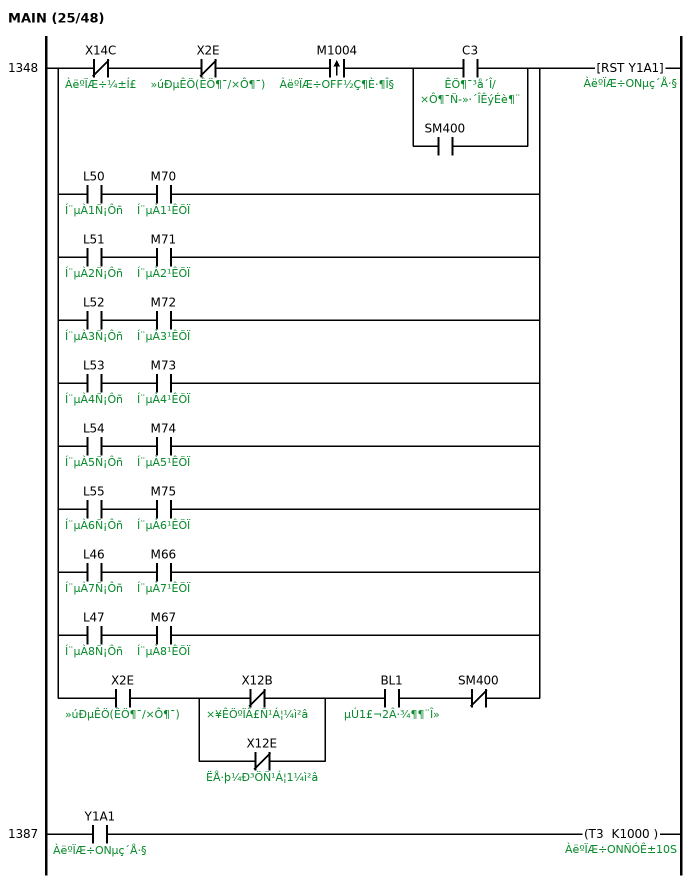
[picture p24: ladder of MAIN, rungs at steps 1348 to 1387]
1348  LDI     X14C  ; ÀëºÏÆ÷¼±Í£
      ANI     X2E  ; »úÐµÊÖ(ÊÖ¶¯/×Ô¶¯)
      ANDP    M1004  ; ÀëºÏÆ÷OFF½Ç¶È·¶Î§
      LD      C3  ; ÊÖ¶¯³å´Î/×Ô¶¯Ñ­»·´ÎÊýÉè¶¨
      OR      SM400
      ANB
      LD      L50  ; Í¨µÀ1Ñ¡Ôñ
      AND     M70  ; Í¨µÀ1¹ÊÕÏ
      ORB
      LD      L51  ; Í¨µÀ2Ñ¡Ôñ
      AND     M71  ; Í¨µÀ2¹ÊÕÏ
      ORB
      LD      L52  ; Í¨µÀ3Ñ¡Ôñ
      AND     M72  ; Í¨µÀ3¹ÊÕÏ
      ORB
      LD      L53  ; Í¨µÀ4Ñ¡Ôñ
      AND     M73  ; Í¨µÀ4¹ÊÕÏ
      ORB
      LD      L54  ; Í¨µÀ5Ñ¡Ôñ
      AND     M74  ; Í¨µÀ5¹ÊÕÏ
      ORB
      LD      L55  ; Í¨µÀ6Ñ¡Ôñ
      AND     M75  ; Í¨µÀ6¹ÊÕÏ
      ORB
      LD      L46  ; Í¨µÀ7Ñ¡Ôñ
      AND     M66  ; Í¨µÀ7¹ÊÕÏ
      ORB
      LD      L47  ; Í¨µÀ8Ñ¡Ôñ
      AND     M67  ; Í¨µÀ8¹ÊÕÏ
      ORB
      LD      X2E  ; »úÐµÊÖ(ÊÖ¶¯/×Ô¶¯)
      LDI     X12B  ; ×¥ÊÖºÏÂ£Ñ¹Á¦¼ì²â
      ORI     X12E  ; ËÅ·þ¼Ð³ÖÑ¹Á¦1¼ì²â
      ANB
      AND     BL1  ; µÚ1£¬2Â·¾¶¶¨Î»
      ANI     SM400
      ORB
      RST     Y1A1  ; ÀëºÏÆ÷ONµç´Å·§
1387  LD      Y1A1  ; ÀëºÏÆ÷ONµç´Å·§
      OUT     T3 K1000  ; ÀëºÏÆ÷ONÑÓÊ±10S
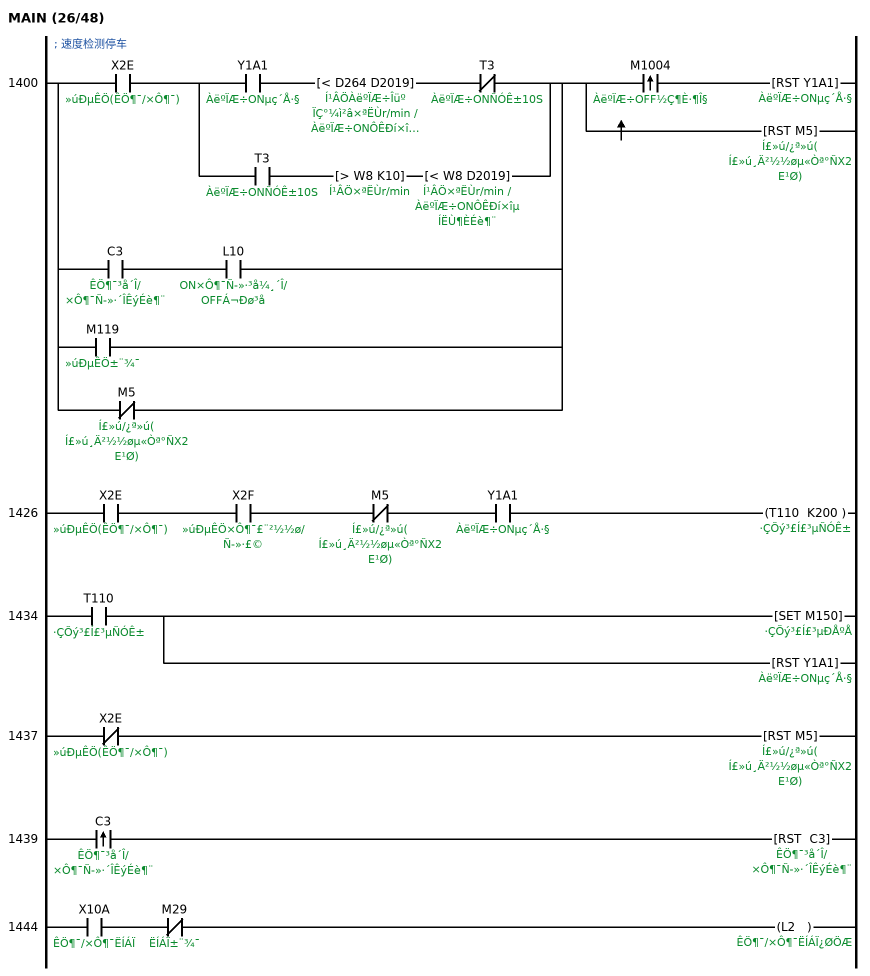
; 速度检测停车
1400  LD      X2E  ; »úÐµÊÖ(ÊÖ¶¯/×Ô¶¯)
      LD      Y1A1  ; ÀëºÏÆ÷ONµç´Å·§
      AND<    D264 D2019  ; Í¹ÂÖÀëºÏÆ÷ÎüºÏÇ°¼ì²â×ªËÙr/min / ÀëºÏÆ÷ONÔÊÐí×îµÍËÙ¶ÈÉè¶¨
      ANI     T3  ; ÀëºÏÆ÷ONÑÓÊ±10S
      LD      T3  ; ÀëºÏÆ÷ONÑÓÊ±10S
      AND>    W8 K10  ; Í¹ÂÖ×ªËÙr/min
      AND<    W8 D2019  ; Í¹ÂÖ×ªËÙr/min / ÀëºÏÆ÷ONÔÊÐí×îµÍËÙ¶ÈÉè¶¨
      ORB
      ANB
      LD      C3  ; ÊÖ¶¯³å´Î/×Ô¶¯Ñ­»·´ÎÊýÉè¶¨
      AND     L10  ; ON×Ô¶¯Ñ­»·³å¼¸´Î/OFFÁ¬Ðø³å
      ORB
      OR      M119  ; »úÐµÊÖ±¨¾¯
      ORI     M5  ; Í£»ú/¿ª»ú(Í£»ú¸Ä²½½øµ«Òª°ÑX2E¹Ø)
      MPS
      ANDP    M1004  ; ÀëºÏÆ÷OFF½Ç¶È·¶Î§
      RST     Y1A1  ; ÀëºÏÆ÷ONµç´Å·§
      MPP
      MEP
      RST     M5  ; Í£»ú/¿ª»ú(Í£»ú¸Ä²½½øµ«Òª°ÑX2E¹Ø)
1426  LD      X2E  ; »úÐµÊÖ(ÊÖ¶¯/×Ô¶¯)
      AND     X2F  ; »úÐµÊÖ×Ô¶¯£¨²½½ø/Ñ­»·£©
      ANI     M5  ; Í£»ú/¿ª»ú(Í£»ú¸Ä²½½øµ«Òª°ÑX2E¹Ø)
      AND     Y1A1  ; ÀëºÏÆ÷ONµç´Å·§
      OUT     T110 K200  ; ·ÇÕý³£Í£³µÑÓÊ±
1434  LD      T110  ; ·ÇÕý³£Í£³µÑÓÊ±
      SET     M150  ; ·ÇÕý³£Í£³µÐÅºÅ
      RST     Y1A1  ; ÀëºÏÆ÷ONµç´Å·§
1437  LDI     X2E  ; »úÐµÊÖ(ÊÖ¶¯/×Ô¶¯)
      RST     M5  ; Í£»ú/¿ª»ú(Í£»ú¸Ä²½½øµ«Òª°ÑX2E¹Ø)
1439  LDP     C3  ; ÊÖ¶¯³å´Î/×Ô¶¯Ñ­»·´ÎÊýÉè¶¨
      RST     C3  ; ÊÖ¶¯³å´Î/×Ô¶¯Ñ­»·´ÎÊýÉè¶¨
1444  LD      X10A  ; ÊÖ¶¯/×Ô¶¯ËÍÁÏ
      ANI     M29  ; ËÍÁÏ±¨¾¯
      OUT     L2  ; ÊÖ¶¯/×Ô¶¯ËÍÁÏ¿ØÖÆ
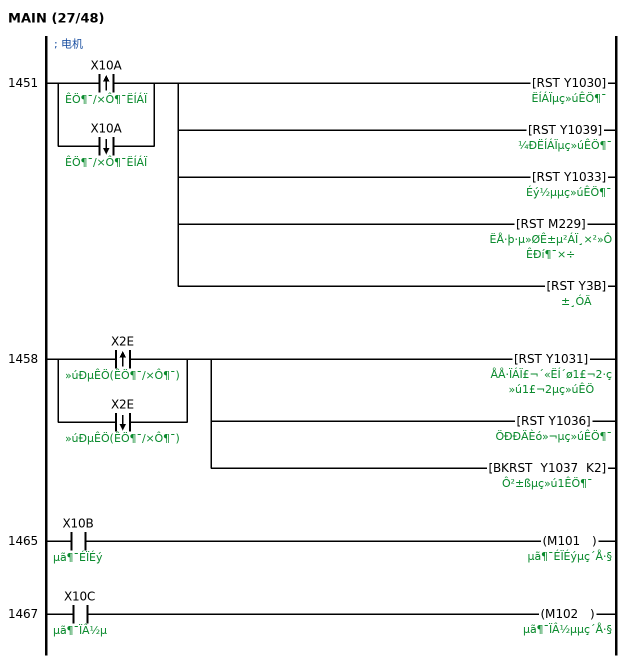
; 电机
1451  LDP     X10A  ; ÊÖ¶¯/×Ô¶¯ËÍÁÏ
      ORF     X10A  ; ÊÖ¶¯/×Ô¶¯ËÍÁÏ
      RST     Y1030  ; ËÍÁÏµç»úÊÖ¶¯
      RST     Y1039  ; ¼ÐËÍÁÏµç»úÊÖ¶¯
      RST     Y1033  ; Éý½µµç»úÊÖ¶¯
      RST     M229  ; ËÅ·þ·µ»ØÊ±µ²ÁÏ¸×²»ÔÊÐí¶¯×÷
      RST     Y3B  ; ±¸ÓÃ
1458  LDP     X2E  ; »úÐµÊÖ(ÊÖ¶¯/×Ô¶¯)
      ORF     X2E  ; »úÐµÊÖ(ÊÖ¶¯/×Ô¶¯)
      RST     Y1031  ; ÅÅ·ÏÁÏ£¬´«ËÍ´ø1£¬2·ç»ú1£¬2µç»úÊÖ
      RST     Y1036  ; ÖÐÐÄÈó»¬µç»úÊÖ¶¯
      BKRST   Y1037 K2  ; Ô²±ßµç»ú1ÊÖ¶¯
1465  LD      X10B  ; µã¶¯ÉÏÉý
      OUT     M101  ; µã¶¯ÉÏÉýµç´Å·§
1467  LD      X10C  ; µã¶¯ÏÂ½µ
      OUT     M102  ; µã¶¯ÏÂ½µµç´Å·§
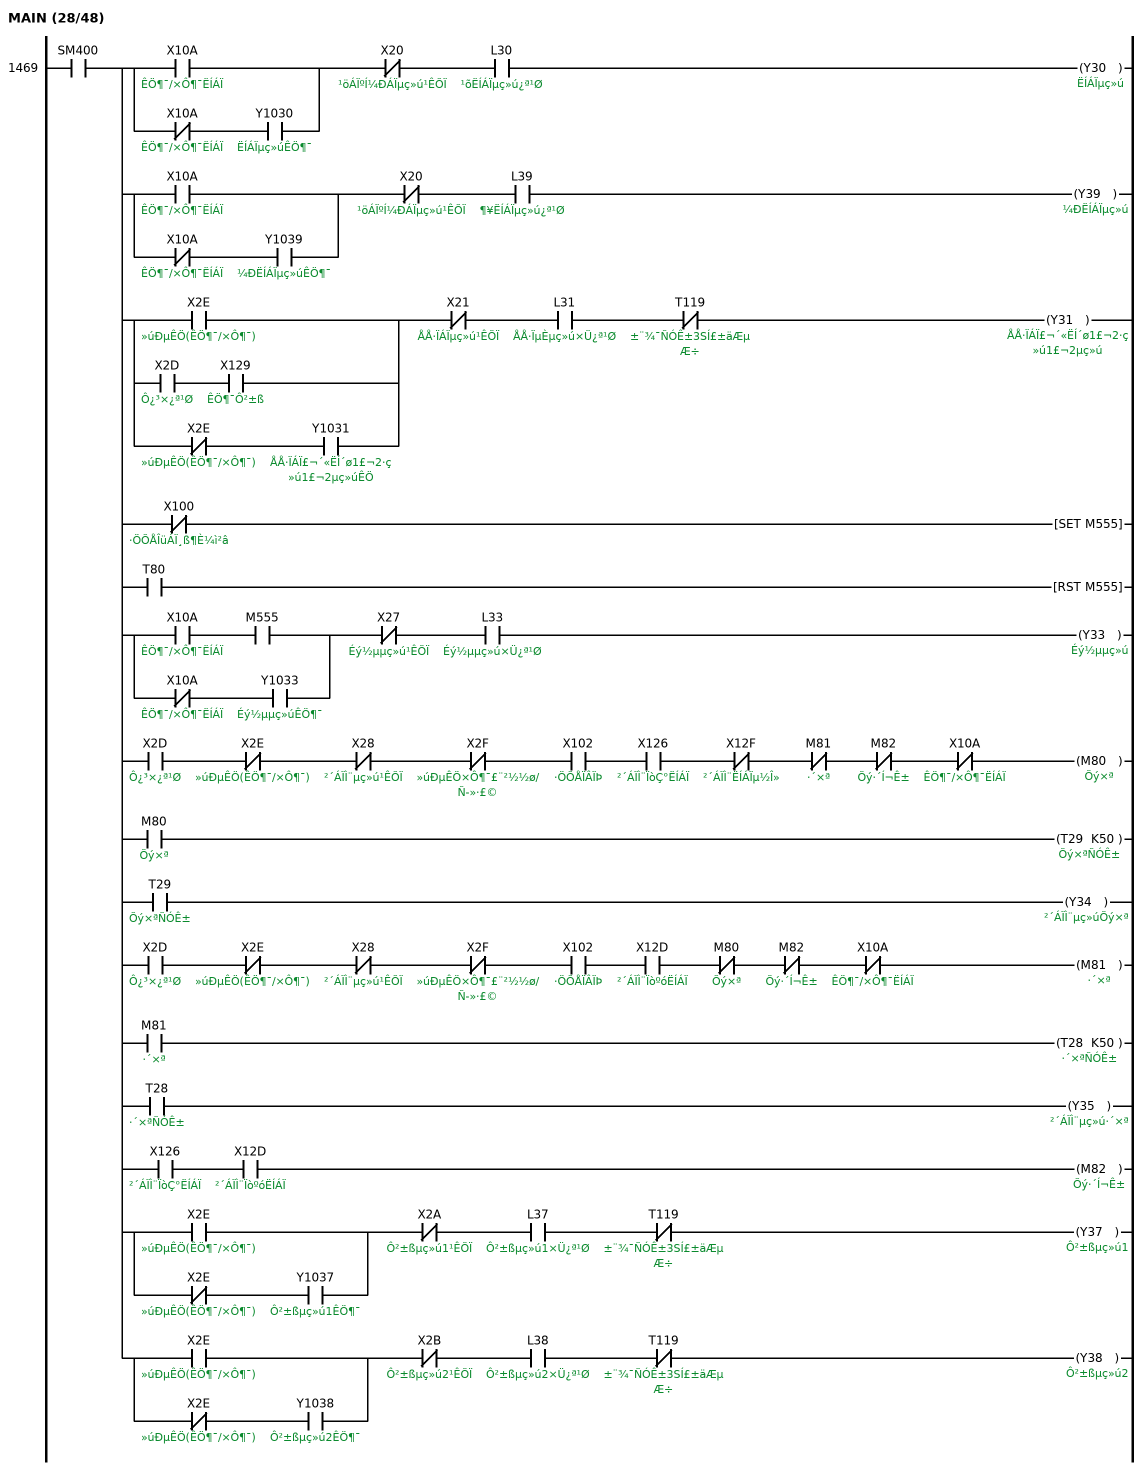
1469  LD      SM400
      MPS
      LD      X10A  ; ÊÖ¶¯/×Ô¶¯ËÍÁÏ
      LDI     X10A  ; ÊÖ¶¯/×Ô¶¯ËÍÁÏ
      AND     Y1030  ; ËÍÁÏµç»úÊÖ¶¯
      ORB
      ANB
      ANI     X20  ; ¹öÁÏºÍ¼ÐÁÏµç»ú¹ÊÕÏ
      AND     L30  ; ¹õËÍÁÏµç»ú¿ª¹Ø
      OUT     Y30  ; ËÍÁÏµç»ú
      MRD
      LD      X10A  ; ÊÖ¶¯/×Ô¶¯ËÍÁÏ
      LDI     X10A  ; ÊÖ¶¯/×Ô¶¯ËÍÁÏ
      AND     Y1039  ; ¼ÐËÍÁÏµç»úÊÖ¶¯
      ORB
      ANB
      ANI     X20  ; ¹öÁÏºÍ¼ÐÁÏµç»ú¹ÊÕÏ
      AND     L39  ; ¶¥ËÍÁÏµç»ú¿ª¹Ø
      OUT     Y39  ; ¼ÐËÍÁÏµç»ú
      MRD
      LD      X2E  ; »úÐµÊÖ(ÊÖ¶¯/×Ô¶¯)
      LD      X2D  ; Ô¿³×¿ª¹Ø
      AND     X129  ; ÊÖ¶¯Ô²±ß
      ORB
      LDI     X2E  ; »úÐµÊÖ(ÊÖ¶¯/×Ô¶¯)
      AND     Y1031  ; ÅÅ·ÏÁÏ£¬´«ËÍ´ø1£¬2·ç»ú1£¬2µç»úÊÖ
      ORB
      ANB
      ANI     X21  ; ÅÅ·ÏÁÏµç»ú¹ÊÕÏ
      AND     L31  ; ÅÅ·ÏµÈµç»ú×Ü¿ª¹Ø
      ANI     T119  ; ±¨¾¯ÑÓÊ±3SÍ£±äÆµÆ÷
      OUT     Y31  ; ÅÅ·ÏÁÏ£¬´«ËÍ´ø1£¬2·ç»ú1£¬2µç»ú
      MRD
      ANI     X100  ; ·ÖÕÅÎüÁÏ¸ß¶È¼ì²â
      SET     M555
      MRD
      AND     T80
      RST     M555
      MRD
      LD      X10A  ; ÊÖ¶¯/×Ô¶¯ËÍÁÏ
      AND     M555
      LDI     X10A  ; ÊÖ¶¯/×Ô¶¯ËÍÁÏ
      AND     Y1033  ; Éý½µµç»úÊÖ¶¯
      ORB
      ANB
      ANI     X27  ; Éý½µµç»ú¹ÊÕÏ
      AND     L33  ; Éý½µµç»ú×Ü¿ª¹Ø
      OUT     Y33  ; Éý½µµç»ú
      MRD
      AND     X2D  ; Ô¿³×¿ª¹Ø
      ANI     X2E  ; »úÐµÊÖ(ÊÖ¶¯/×Ô¶¯)
      ANI     X28  ; ²´ÁÏÌ¨µç»ú¹ÊÕÏ
      ANI     X2F  ; »úÐµÊÖ×Ô¶¯£¨²½½ø/Ñ­»·£©
      AND     X102  ; ·ÖÕÅÏÂÏÞ
      AND     X126  ; ²´ÁÏÌ¨ÏòÇ°ËÍÁÏ
      ANI     X12F  ; ²´ÁÏÌ¨ËÍÁÏµ½Î»
      ANI     M81  ; ·´×ª
      ANI     M82  ; Õý·´Í¬Ê±
      ANI     X10A  ; ÊÖ¶¯/×Ô¶¯ËÍÁÏ
      OUT     M80  ; Õý×ª
      MRD
      AND     M80  ; Õý×ª
      OUT     T29 K50  ; Õý×ªÑÓÊ±
      MRD
      AND     T29  ; Õý×ªÑÓÊ±
      OUT     Y34  ; ²´ÁÏÌ¨µç»úÕý×ª
      MRD
      AND     X2D  ; Ô¿³×¿ª¹Ø
      ANI     X2E  ; »úÐµÊÖ(ÊÖ¶¯/×Ô¶¯)
      ANI     X28  ; ²´ÁÏÌ¨µç»ú¹ÊÕÏ
      ANI     X2F  ; »úÐµÊÖ×Ô¶¯£¨²½½ø/Ñ­»·£©
      AND     X102  ; ·ÖÕÅÏÂÏÞ
      AND     X12D  ; ²´ÁÏÌ¨ÏòºóËÍÁÏ
      ANI     M80  ; Õý×ª
      ANI     M82  ; Õý·´Í¬Ê±
      ANI     X10A  ; ÊÖ¶¯/×Ô¶¯ËÍÁÏ
      OUT     M81  ; ·´×ª
      MRD
      AND     M81  ; ·´×ª
      OUT     T28 K50  ; ·´×ªÑÓÊ±
      MRD
      AND     T28  ; ·´×ªÑÓÊ±
      OUT     Y35  ; ²´ÁÏÌ¨µç»ú·´×ª
      MRD
      AND     X126  ; ²´ÁÏÌ¨ÏòÇ°ËÍÁÏ
      AND     X12D  ; ²´ÁÏÌ¨ÏòºóËÍÁÏ
      OUT     M82  ; Õý·´Í¬Ê±
      MRD
      LD      X2E  ; »úÐµÊÖ(ÊÖ¶¯/×Ô¶¯)
      LDI     X2E  ; »úÐµÊÖ(ÊÖ¶¯/×Ô¶¯)
      AND     Y1037  ; Ô²±ßµç»ú1ÊÖ¶¯
      ORB
      ANB
      ANI     X2A  ; Ô²±ßµç»ú1¹ÊÕÏ
      AND     L37  ; Ô²±ßµç»ú1×Ü¿ª¹Ø
      ANI     T119  ; ±¨¾¯ÑÓÊ±3SÍ£±äÆµÆ÷
      OUT     Y37  ; Ô²±ßµç»ú1
      MPP
      LD      X2E  ; »úÐµÊÖ(ÊÖ¶¯/×Ô¶¯)
      LDI     X2E  ; »úÐµÊÖ(ÊÖ¶¯/×Ô¶¯)
      AND     Y1038  ; Ô²±ßµç»ú2ÊÖ¶¯
      ORB
      ANB
      ANI     X2B  ; Ô²±ßµç»ú2¹ÊÕÏ
      AND     L38  ; Ô²±ßµç»ú2×Ü¿ª¹Ø
      ANI     T119  ; ±¨¾¯ÑÓÊ±3SÍ£±äÆµÆ÷
      OUT     Y38  ; Ô²±ßµç»ú2
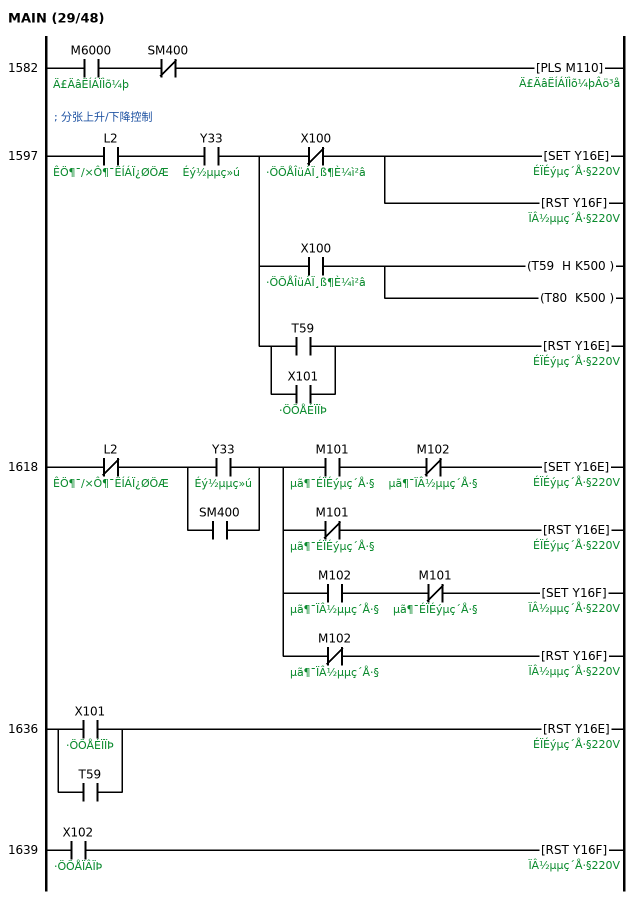
1582  LD      M6000  ; Ä£ÄâËÍÁÏÌõ¼þ
      ANI     SM400
      PLS     M110  ; Ä£ÄâËÍÁÏÌõ¼þÂö³å
; 分张上升/下降控制
1597  LD      L2  ; ÊÖ¶¯/×Ô¶¯ËÍÁÏ¿ØÖÆ
      AND     Y33  ; Éý½µµç»ú
      MPS
      ANI     X100  ; ·ÖÕÅÎüÁÏ¸ß¶È¼ì²â
      SET     Y16E  ; ÉÏÉýµç´Å·§220V
      RST     Y16F  ; ÏÂ½µµç´Å·§220V
      MRD
      AND     X100  ; ·ÖÕÅÎüÁÏ¸ß¶È¼ì²â
      OUTH    T59 K500
      OUT     T80 K500
      MPP
      LD      T59
      OR      X101  ; ·ÖÕÅÉÏÏÞ
      ANB
      RST     Y16E  ; ÉÏÉýµç´Å·§220V
1618  LDI     L2  ; ÊÖ¶¯/×Ô¶¯ËÍÁÏ¿ØÖÆ
      LD      Y33  ; Éý½µµç»ú
      OR      SM400
      ANB
      MPS
      AND     M101  ; µã¶¯ÉÏÉýµç´Å·§
      ANI     M102  ; µã¶¯ÏÂ½µµç´Å·§
      SET     Y16E  ; ÉÏÉýµç´Å·§220V
      MRD
      ANI     M101  ; µã¶¯ÉÏÉýµç´Å·§
      RST     Y16E  ; ÉÏÉýµç´Å·§220V
      MRD
      AND     M102  ; µã¶¯ÏÂ½µµç´Å·§
      ANI     M101  ; µã¶¯ÉÏÉýµç´Å·§
      SET     Y16F  ; ÏÂ½µµç´Å·§220V
      MPP
      ANI     M102  ; µã¶¯ÏÂ½µµç´Å·§
      RST     Y16F  ; ÏÂ½µµç´Å·§220V
1636  LD      X101  ; ·ÖÕÅÉÏÏÞ
      OR      T59
      RST     Y16E  ; ÉÏÉýµç´Å·§220V
1639  LD      X102  ; ·ÖÕÅÏÂÏÞ
      RST     Y16F  ; ÏÂ½µµç´Å·§220V
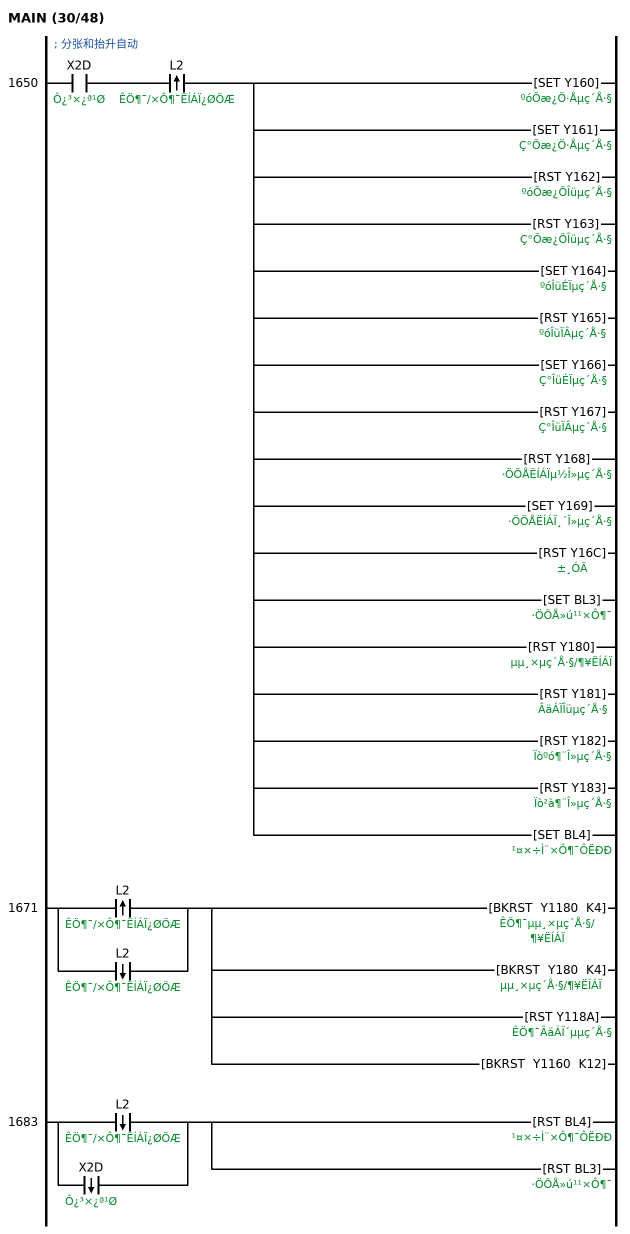
; 分张和抬升自动
1650  LD      X2D  ; Ô¿³×¿ª¹Ø
      ANDP    L2  ; ÊÖ¶¯/×Ô¶¯ËÍÁÏ¿ØÖÆ
      SET     Y160  ; ºóÕæ¿Õ·Åµç´Å·§
      SET     Y161  ; Ç°Õæ¿Õ·Åµç´Å·§
      RST     Y162  ; ºóÕæ¿ÕÎüµç´Å·§
      RST     Y163  ; Ç°Õæ¿ÕÎüµç´Å·§
      SET     Y164  ; ºóÎüÉÏµç´Å·§
      RST     Y165  ; ºóÎüÏÂµç´Å·§
      SET     Y166  ; Ç°ÎüÉÏµç´Å·§
      RST     Y167  ; Ç°ÎüÏÂµç´Å·§
      RST     Y168  ; ·ÖÕÅËÍÁÏµ½Î»µç´Å·§
      SET     Y169  ; ·ÖÕÅËÍÁÏ¸´Î»µç´Å·§
      RST     Y16C  ; ±¸ÓÃ
      SET     BL3  ; ·ÖÕÅ»ú¹¹×Ô¶¯
      RST     Y180  ; µµ¸×µç´Å·§/¶¥ËÍÁÏ
      RST     Y181  ; ÂäÁÏÎüµç´Å·§
      RST     Y182  ; Ïòºó¶¨Î»µç´Å·§
      RST     Y183  ; Ïò²à¶¨Î»µç´Å·§
      SET     BL4  ; ¹¤×÷Ì¨×Ô¶¯ÔËÐÐ
1671  LDP     L2  ; ÊÖ¶¯/×Ô¶¯ËÍÁÏ¿ØÖÆ
      ORF     L2  ; ÊÖ¶¯/×Ô¶¯ËÍÁÏ¿ØÖÆ
      BKRST   Y1180 K4  ; ÊÖ¶¯µµ¸×µç´Å·§/¶¥ËÍÁÏ
      BKRST   Y180 K4
      RST     Y118A  ; ÊÖ¶¯ÂäÁÏ´µµç´Å·§
      BKRST   Y1160 K12
1683  LDF     L2  ; ÊÖ¶¯/×Ô¶¯ËÍÁÏ¿ØÖÆ
      ORF     X2D  ; Ô¿³×¿ª¹Ø
      RST     BL4  ; ¹¤×÷Ì¨×Ô¶¯ÔËÐÐ
      RST     BL3  ; ·ÖÕÅ»ú¹¹×Ô¶¯
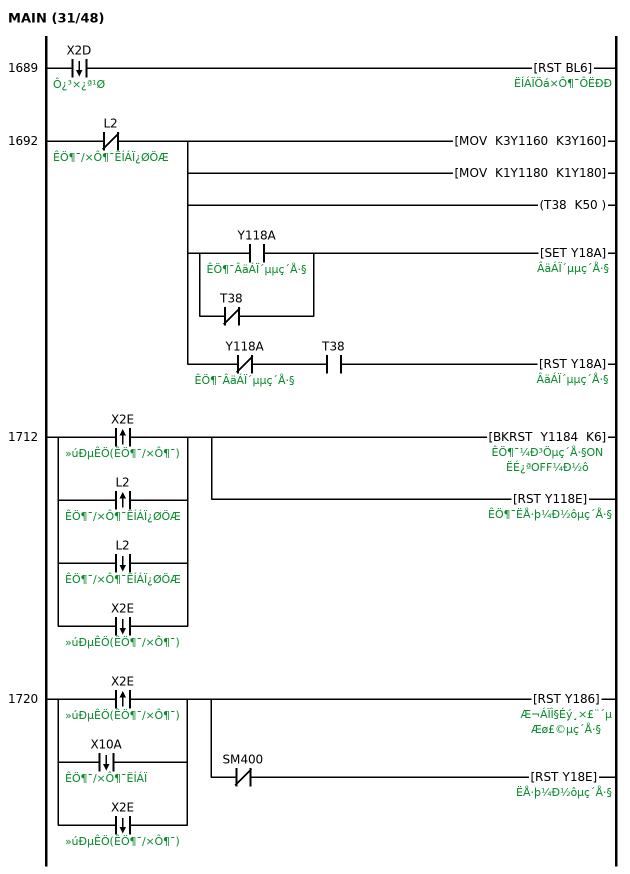
1689  LDF     X2D  ; Ô¿³×¿ª¹Ø
      RST     BL6  ; ËÍÁÏÖá×Ô¶¯ÔËÐÐ
1692  LDI     L2  ; ÊÖ¶¯/×Ô¶¯ËÍÁÏ¿ØÖÆ
      MOV     K3Y1160 K3Y160
      MOV     K1Y1180 K1Y180
      OUT     T38 K50
      MPS
      LD      Y118A  ; ÊÖ¶¯ÂäÁÏ´µµç´Å·§
      ORI     T38
      ANB
      SET     Y18A  ; ÂäÁÏ´µµç´Å·§
      MPP
      ANI     Y118A  ; ÊÖ¶¯ÂäÁÏ´µµç´Å·§
      AND     T38
      RST     Y18A  ; ÂäÁÏ´µµç´Å·§
1712  LDP     X2E  ; »úÐµÊÖ(ÊÖ¶¯/×Ô¶¯)
      ORP     L2  ; ÊÖ¶¯/×Ô¶¯ËÍÁÏ¿ØÖÆ
      ORF     L2  ; ÊÖ¶¯/×Ô¶¯ËÍÁÏ¿ØÖÆ
      ORF     X2E  ; »úÐµÊÖ(ÊÖ¶¯/×Ô¶¯)
      BKRST   Y1184 K6  ; ÊÖ¶¯¼Ð³Öµç´Å·§ONËÉ¿ªOFF¼Ð½ô
      RST     Y118E  ; ÊÖ¶¯ËÅ·þ¼Ð½ôµç´Å·§
1720  LDP     X2E  ; »úÐµÊÖ(ÊÖ¶¯/×Ô¶¯)
      ORF     X10A  ; ÊÖ¶¯/×Ô¶¯ËÍÁÏ
      ORF     X2E  ; »úÐµÊÖ(ÊÖ¶¯/×Ô¶¯)
      RST     Y186  ; Æ¬ÁÏÌ§Éý¸×£¨´µÆø£©µç´Å·§
      ANI     SM400
      RST     Y18E  ; ËÅ·þ¼Ð½ôµç´Å·§
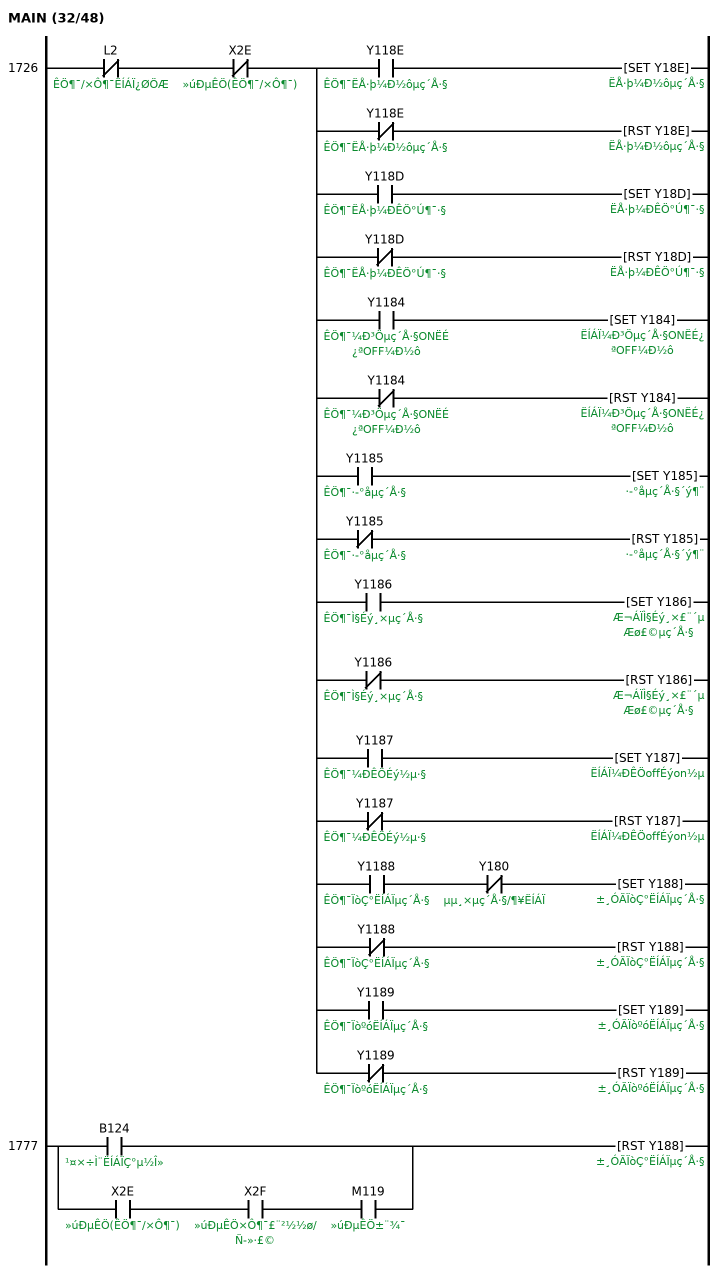
1726  LDI     L2  ; ÊÖ¶¯/×Ô¶¯ËÍÁÏ¿ØÖÆ
      ANI     X2E  ; »úÐµÊÖ(ÊÖ¶¯/×Ô¶¯)
      MPS
      AND     Y118E  ; ÊÖ¶¯ËÅ·þ¼Ð½ôµç´Å·§
      SET     Y18E  ; ËÅ·þ¼Ð½ôµç´Å·§
      MRD
      ANI     Y118E  ; ÊÖ¶¯ËÅ·þ¼Ð½ôµç´Å·§
      RST     Y18E  ; ËÅ·þ¼Ð½ôµç´Å·§
      MRD
      AND     Y118D  ; ÊÖ¶¯ËÅ·þ¼ÐÊÖ°Ú¶¯·§
      SET     Y18D  ; ËÅ·þ¼ÐÊÖ°Ú¶¯·§
      MRD
      ANI     Y118D  ; ÊÖ¶¯ËÅ·þ¼ÐÊÖ°Ú¶¯·§
      RST     Y18D  ; ËÅ·þ¼ÐÊÖ°Ú¶¯·§
      MRD
      AND     Y1184  ; ÊÖ¶¯¼Ð³Öµç´Å·§ONËÉ¿ªOFF¼Ð½ô
      SET     Y184  ; ËÍÁÏ¼Ð³Öµç´Å·§ONËÉ¿ªOFF¼Ð½ô
      MRD
      ANI     Y1184  ; ÊÖ¶¯¼Ð³Öµç´Å·§ONËÉ¿ªOFF¼Ð½ô
      RST     Y184  ; ËÍÁÏ¼Ð³Öµç´Å·§ONËÉ¿ªOFF¼Ð½ô
      MRD
      AND     Y1185  ; ÊÖ¶¯·­°åµç´Å·§
      SET     Y185  ; ·­°åµç´Å·§´ý¶¨
      MRD
      ANI     Y1185  ; ÊÖ¶¯·­°åµç´Å·§
      RST     Y185  ; ·­°åµç´Å·§´ý¶¨
      MRD
      AND     Y1186  ; ÊÖ¶¯Ì§Éý¸×µç´Å·§
      SET     Y186  ; Æ¬ÁÏÌ§Éý¸×£¨´µÆø£©µç´Å·§
      MRD
      ANI     Y1186  ; ÊÖ¶¯Ì§Éý¸×µç´Å·§
      RST     Y186  ; Æ¬ÁÏÌ§Éý¸×£¨´µÆø£©µç´Å·§
      MRD
      AND     Y1187  ; ÊÖ¶¯¼ÐÊÖÉý½µ·§
      SET     Y187  ; ËÍÁÏ¼ÐÊÖoffÉýon½µ
      MRD
      ANI     Y1187  ; ÊÖ¶¯¼ÐÊÖÉý½µ·§
      RST     Y187  ; ËÍÁÏ¼ÐÊÖoffÉýon½µ
      MRD
      AND     Y1188  ; ÊÖ¶¯ÏòÇ°ËÍÁÏµç´Å·§
      ANI     Y180  ; µµ¸×µç´Å·§/¶¥ËÍÁÏ
      SET     Y188  ; ±¸ÓÃÏòÇ°ËÍÁÏµç´Å·§
      MRD
      ANI     Y1188  ; ÊÖ¶¯ÏòÇ°ËÍÁÏµç´Å·§
      RST     Y188  ; ±¸ÓÃÏòÇ°ËÍÁÏµç´Å·§
      MRD
      AND     Y1189  ; ÊÖ¶¯ÏòºóËÍÁÏµç´Å·§
      SET     Y189  ; ±¸ÓÃÏòºóËÍÁÏµç´Å·§
      MPP
      ANI     Y1189  ; ÊÖ¶¯ÏòºóËÍÁÏµç´Å·§
      RST     Y189  ; ±¸ÓÃÏòºóËÍÁÏµç´Å·§
1777  LD      B124  ; ¹¤×÷Ì¨ËÍÁÏÇ°µ½Î»
      LD      X2E  ; »úÐµÊÖ(ÊÖ¶¯/×Ô¶¯)
      AND     X2F  ; »úÐµÊÖ×Ô¶¯£¨²½½ø/Ñ­»·£©
      AND     M119  ; »úÐµÊÖ±¨¾¯
      ORB
      RST     Y188  ; ±¸ÓÃÏòÇ°ËÍÁÏµç´Å·§
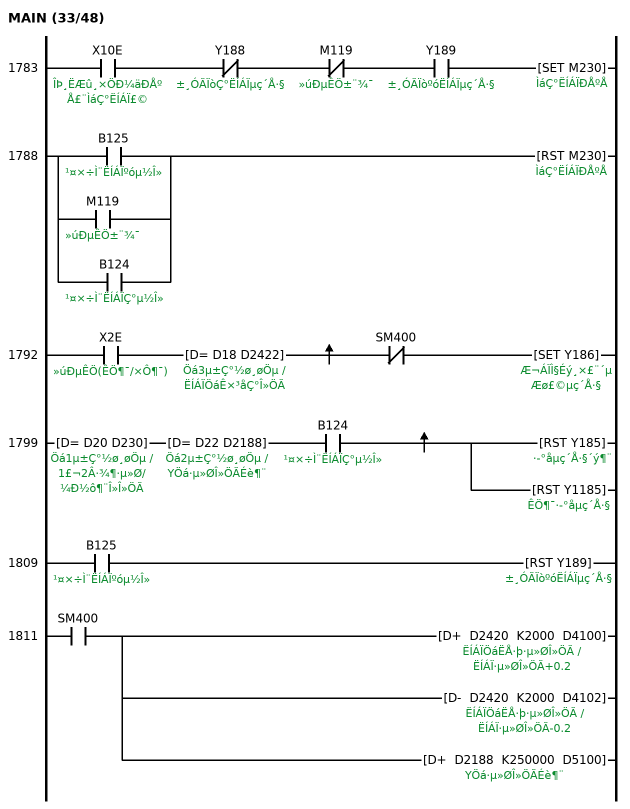
1783  LD      X10E  ; ÎÞ¸ËÆû¸×ÖÐ¼äÐÅºÅ£¨ÌáÇ°ËÍÁÏ£©
      ANI     Y188  ; ±¸ÓÃÏòÇ°ËÍÁÏµç´Å·§
      ANI     M119  ; »úÐµÊÖ±¨¾¯
      AND     Y189  ; ±¸ÓÃÏòºóËÍÁÏµç´Å·§
      SET     M230  ; ÌáÇ°ËÍÁÏÐÅºÅ
1788  LD      B125  ; ¹¤×÷Ì¨ËÍÁÏºóµ½Î»
      OR      M119  ; »úÐµÊÖ±¨¾¯
      OR      B124  ; ¹¤×÷Ì¨ËÍÁÏÇ°µ½Î»
      RST     M230  ; ÌáÇ°ËÍÁÏÐÅºÅ
1792  LD      X2E  ; »úÐµÊÖ(ÊÖ¶¯/×Ô¶¯)
      ANDD=   D18 D2422  ; Öá3µ±Ç°½ø¸øÖµ / ËÍÁÏÖáÊ×³åÇ°Î»ÖÃ
      MEP
      ANI     SM400
      SET     Y186  ; Æ¬ÁÏÌ§Éý¸×£¨´µÆø£©µç´Å·§
1799  LDD=    D20 D230  ; Öá1µ±Ç°½ø¸øÖµ / 1£¬2Â·¾¶·µ»Ø/¼Ð½ô¶¨Î»Î»ÖÃ
      ANDD=   D22 D2188  ; Öá2µ±Ç°½ø¸øÖµ / YÖá·µ»ØÎ»ÖÃÉè¶¨
      AND     B124  ; ¹¤×÷Ì¨ËÍÁÏÇ°µ½Î»
      MEP
      RST     Y185  ; ·­°åµç´Å·§´ý¶¨
      RST     Y1185  ; ÊÖ¶¯·­°åµç´Å·§
1809  LD      B125  ; ¹¤×÷Ì¨ËÍÁÏºóµ½Î»
      RST     Y189  ; ±¸ÓÃÏòºóËÍÁÏµç´Å·§
1811  LD      SM400
      D+      D2420 K2000 D4100  ; ËÍÁÏ·µ»ØÎ»ÖÃ+0.2
      D-      D2420 K2000 D4102  ; ËÍÁÏ·µ»ØÎ»ÖÃ-0.2
      D+      D2188 K250000 D5100
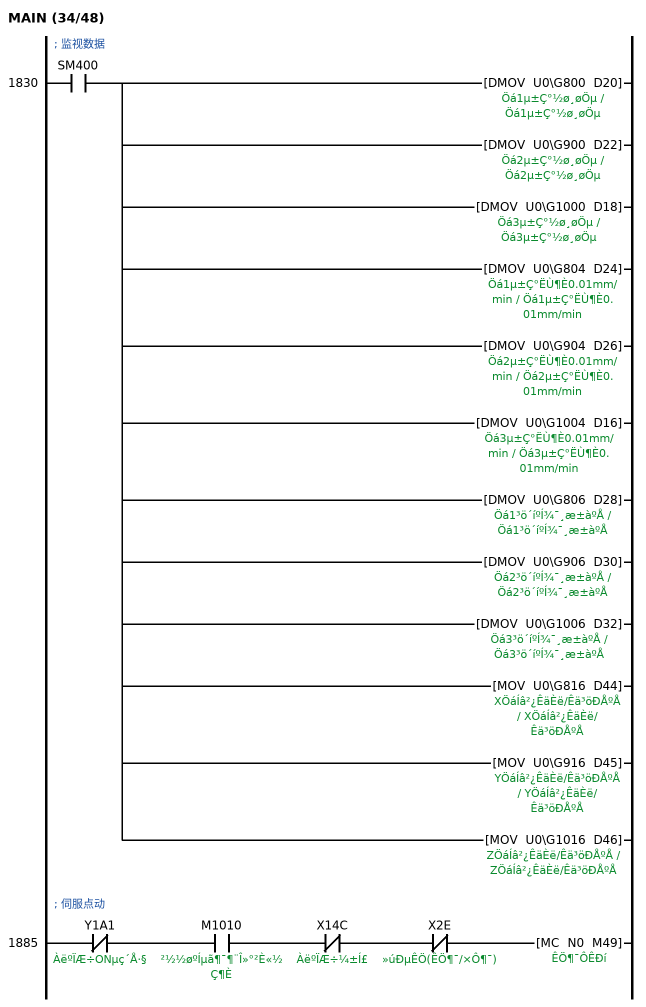
; 监视数据
1830  LD      SM400
      DMOV    U0\G800 D20  ; Öá1µ±Ç°½ø¸øÖµ
      DMOV    U0\G900 D22  ; Öá2µ±Ç°½ø¸øÖµ
      DMOV    U0\G1000 D18  ; Öá3µ±Ç°½ø¸øÖµ
      DMOV    U0\G804 D24  ; Öá1µ±Ç°ËÙ¶È0.01mm/min / Öá1µ±Ç°ËÙ¶È0.01mm/min
      DMOV    U0\G904 D26  ; Öá2µ±Ç°ËÙ¶È0.01mm/min / Öá2µ±Ç°ËÙ¶È0.01mm/min
      DMOV    U0\G1004 D16  ; Öá3µ±Ç°ËÙ¶È0.01mm/min / Öá3µ±Ç°ËÙ¶È0.01mm/min
      DMOV    U0\G806 D28  ; Öá1³ö´íºÍ¾¯¸æ±àºÅ
      DMOV    U0\G906 D30  ; Öá2³ö´íºÍ¾¯¸æ±àºÅ
      DMOV    U0\G1006 D32  ; Öá3³ö´íºÍ¾¯¸æ±àºÅ / Öá3³ö´íºÍ¾¯¸æ±àºÅ
      MOV     U0\G816 D44  ; XÖáÍâ²¿ÊäÈë/Êä³öÐÅºÅ / XÖáÍâ²¿ÊäÈë/Êä³öÐÅºÅ
      MOV     U0\G916 D45  ; YÖáÍâ²¿ÊäÈë/Êä³öÐÅºÅ / YÖáÍâ²¿ÊäÈë/Êä³öÐÅºÅ
      MOV     U0\G1016 D46  ; ZÖáÍâ²¿ÊäÈë/Êä³öÐÅºÅ / ZÖáÍâ²¿ÊäÈë/Êä³öÐÅºÅ
; 伺服点动
1885  LDI     Y1A1  ; ÀëºÏÆ÷ONµç´Å·§
      AND     M1010  ; ²½½øºÍµã¶¯¶¨Î»°²È«½Ç¶È
      ANI     X14C  ; ÀëºÏÆ÷¼±Í£
      ANI     X2E  ; »úÐµÊÖ(ÊÖ¶¯/×Ô¶¯)
      MC      N0 M49  ; ÊÖ¶¯ÔÊÐí
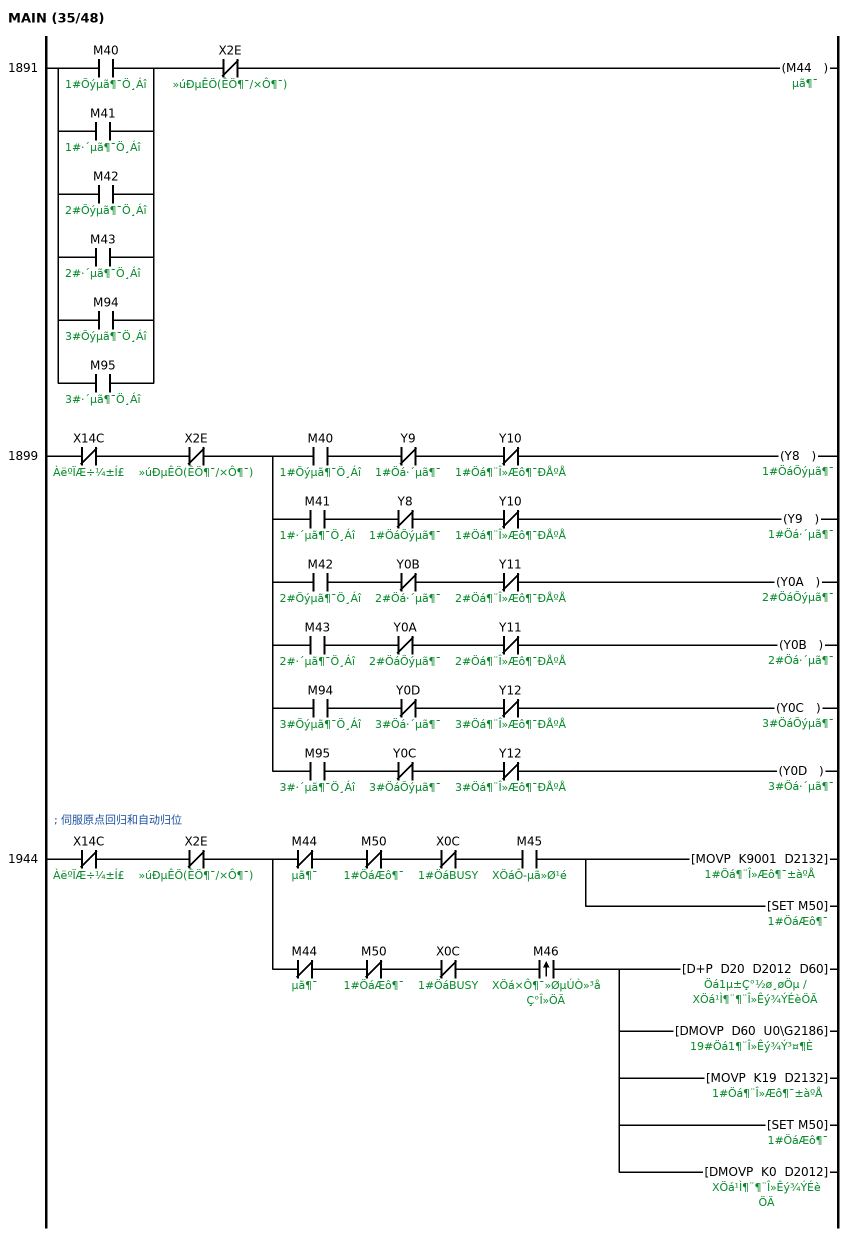
1891  LD      M40  ; 1#Õýµã¶¯Ö¸Áî
      OR      M41  ; 1#·´µã¶¯Ö¸Áî
      OR      M42  ; 2#Õýµã¶¯Ö¸Áî
      OR      M43  ; 2#·´µã¶¯Ö¸Áî
      OR      M94  ; 3#Õýµã¶¯Ö¸Áî
      OR      M95  ; 3#·´µã¶¯Ö¸Áî
      ANI     X2E  ; »úÐµÊÖ(ÊÖ¶¯/×Ô¶¯)
      OUT     M44  ; µã¶¯
1899  LDI     X14C  ; ÀëºÏÆ÷¼±Í£
      ANI     X2E  ; »úÐµÊÖ(ÊÖ¶¯/×Ô¶¯)
      MPS
      AND     M40  ; 1#Õýµã¶¯Ö¸Áî
      ANI     Y9  ; 1#Öá·´µã¶¯
      ANI     Y10  ; 1#Öá¶¨Î»Æô¶¯ÐÅºÅ
      OUT     Y8  ; 1#ÖáÕýµã¶¯
      MRD
      AND     M41  ; 1#·´µã¶¯Ö¸Áî
      ANI     Y8  ; 1#ÖáÕýµã¶¯
      ANI     Y10  ; 1#Öá¶¨Î»Æô¶¯ÐÅºÅ
      OUT     Y9  ; 1#Öá·´µã¶¯
      MRD
      AND     M42  ; 2#Õýµã¶¯Ö¸Áî
      ANI     Y0B  ; 2#Öá·´µã¶¯
      ANI     Y11  ; 2#Öá¶¨Î»Æô¶¯ÐÅºÅ
      OUT     Y0A  ; 2#ÖáÕýµã¶¯
      MRD
      AND     M43  ; 2#·´µã¶¯Ö¸Áî
      ANI     Y0A  ; 2#ÖáÕýµã¶¯
      ANI     Y11  ; 2#Öá¶¨Î»Æô¶¯ÐÅºÅ
      OUT     Y0B  ; 2#Öá·´µã¶¯
      MRD
      AND     M94  ; 3#Õýµã¶¯Ö¸Áî
      ANI     Y0D  ; 3#Öá·´µã¶¯
      ANI     Y12  ; 3#Öá¶¨Î»Æô¶¯ÐÅºÅ
      OUT     Y0C  ; 3#ÖáÕýµã¶¯
      MPP
      AND     M95  ; 3#·´µã¶¯Ö¸Áî
      ANI     Y0C  ; 3#ÖáÕýµã¶¯
      ANI     Y12  ; 3#Öá¶¨Î»Æô¶¯ÐÅºÅ
      OUT     Y0D  ; 3#Öá·´µã¶¯
; 伺服原点回归和自动归位
1944  LDI     X14C  ; ÀëºÏÆ÷¼±Í£
      ANI     X2E  ; »úÐµÊÖ(ÊÖ¶¯/×Ô¶¯)
      MPS
      ANI     M44  ; µã¶¯
      ANI     M50  ; 1#ÖáÆô¶¯
      ANI     X0C  ; 1#ÖáBUSY
      AND     M45  ; XÖáÔ­µã»Ø¹é
      MOVP    K9001 D2132  ; 1#Öá¶¨Î»Æô¶¯±àºÅ
      SET     M50  ; 1#ÖáÆô¶¯
      MPP
      ANI     M44  ; µã¶¯
      ANI     M50  ; 1#ÖáÆô¶¯
      ANI     X0C  ; 1#ÖáBUSY
      ANDP    M46  ; XÖá×Ô¶¯»ØµÚÒ»³åÇ°Î»ÖÃ
      D+P     D20 D2012 D60  ; XÖá¹Ì¶¨¶¨Î»Êý¾ÝÉèÖÃ
      DMOVP   D60 U0\G2186  ; 19#Öá1¶¨Î»Êý¾Ý³¤¶È
      MOVP    K19 D2132
      SET     M50  ; 1#ÖáÆô¶¯
      DMOVP   K0 D2012
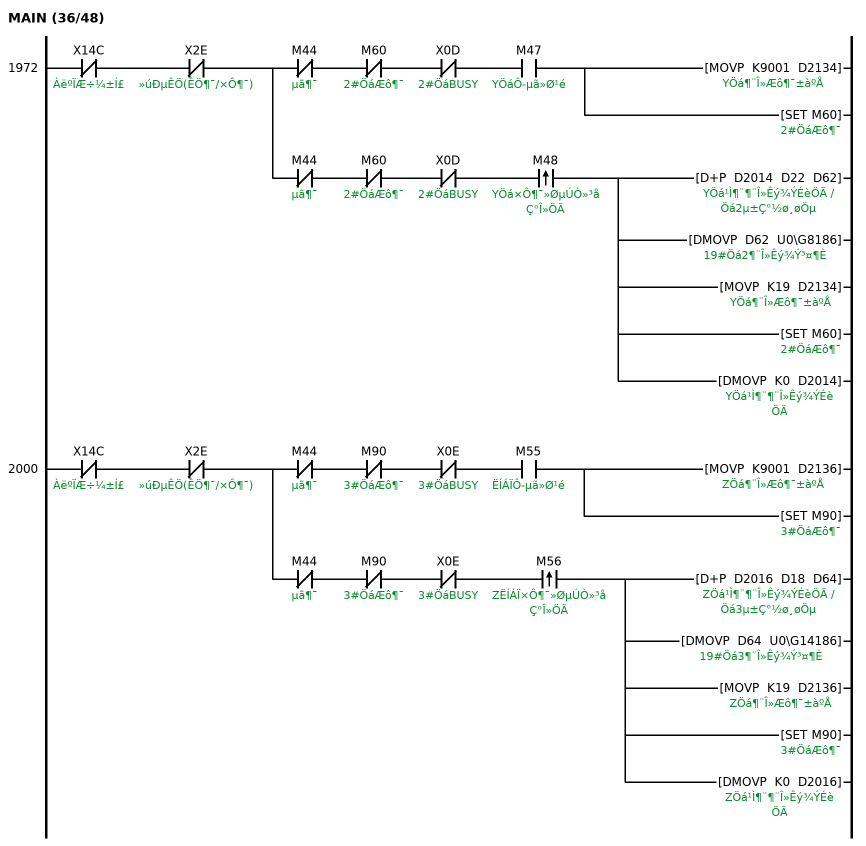
1972  LDI     X14C  ; ÀëºÏÆ÷¼±Í£
      ANI     X2E  ; »úÐµÊÖ(ÊÖ¶¯/×Ô¶¯)
      MPS
      ANI     M44  ; µã¶¯
      ANI     M60  ; 2#ÖáÆô¶¯
      ANI     X0D  ; 2#ÖáBUSY
      AND     M47  ; YÖáÔ­µã»Ø¹é
      MOVP    K9001 D2134  ; YÖá¶¨Î»Æô¶¯±àºÅ
      SET     M60  ; 2#ÖáÆô¶¯
      MPP
      ANI     M44  ; µã¶¯
      ANI     M60  ; 2#ÖáÆô¶¯
      ANI     X0D  ; 2#ÖáBUSY
      ANDP    M48  ; YÖá×Ô¶¯»ØµÚÒ»³åÇ°Î»ÖÃ
      D+P     D2014 D22 D62  ; YÖá¹Ì¶¨¶¨Î»Êý¾ÝÉèÖÃ
      DMOVP   D62 U0\G8186  ; 19#Öá2¶¨Î»Êý¾Ý³¤¶È
      MOVP    K19 D2134
      SET     M60  ; 2#ÖáÆô¶¯
      DMOVP   K0 D2014
2000  LDI     X14C  ; ÀëºÏÆ÷¼±Í£
      ANI     X2E  ; »úÐµÊÖ(ÊÖ¶¯/×Ô¶¯)
      MPS
      ANI     M44  ; µã¶¯
      ANI     M90  ; 3#ÖáÆô¶¯
      ANI     X0E  ; 3#ÖáBUSY
      AND     M55  ; ËÍÁÏÔ­µã»Ø¹é
      MOVP    K9001 D2136  ; ZÖá¶¨Î»Æô¶¯±àºÅ
      SET     M90  ; 3#ÖáÆô¶¯
      MPP
      ANI     M44  ; µã¶¯
      ANI     M90  ; 3#ÖáÆô¶¯
      ANI     X0E  ; 3#ÖáBUSY
      ANDP    M56  ; ZËÍÁÏ×Ô¶¯»ØµÚÒ»³åÇ°Î»ÖÃ
      D+P     D2016 D18 D64  ; ZÖá¹Ì¶¨¶¨Î»Êý¾ÝÉèÖÃ
      DMOVP   D64 U0\G14186  ; 19#Öá3¶¨Î»Êý¾Ý³¤¶È
      MOVP    K19 D2136
      SET     M90  ; 3#ÖáÆô¶¯
      DMOVP   K0 D2016
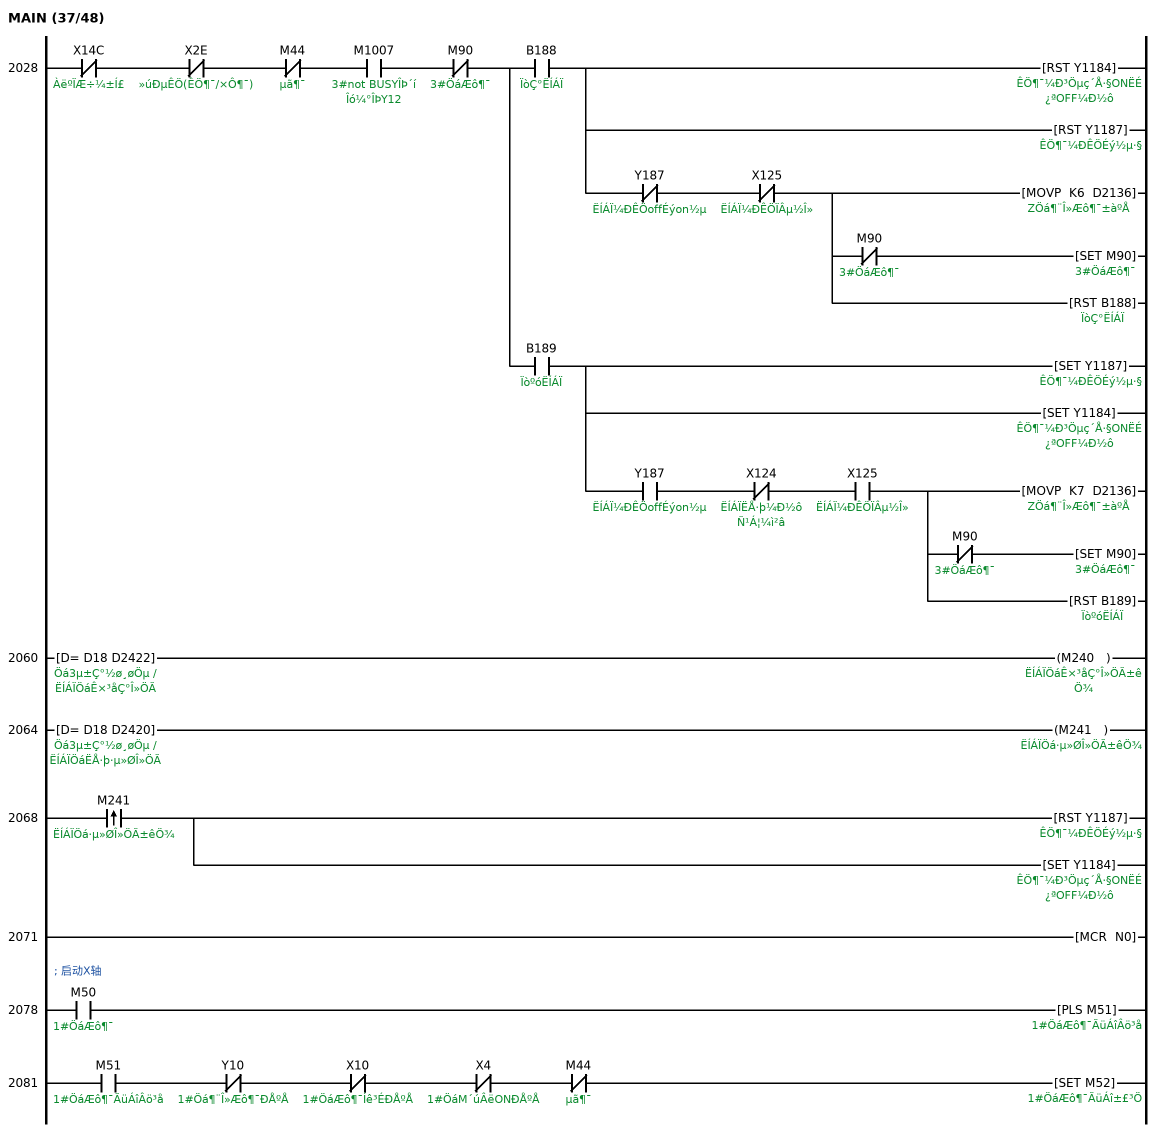
2028  LDI     X14C  ; ÀëºÏÆ÷¼±Í£
      ANI     X2E  ; »úÐµÊÖ(ÊÖ¶¯/×Ô¶¯)
      ANI     M44  ; µã¶¯
      AND     M1007  ; 3#not BUSYÎÞ´íÎó¼°ÎÞY12
      ANI     M90  ; 3#ÖáÆô¶¯
      MPS
      AND     B188  ; ÏòÇ°ËÍÁÏ
      RST     Y1184  ; ÊÖ¶¯¼Ð³Öµç´Å·§ONËÉ¿ªOFF¼Ð½ô
      RST     Y1187  ; ÊÖ¶¯¼ÐÊÖÉý½µ·§
      ANI     Y187  ; ËÍÁÏ¼ÐÊÖoffÉýon½µ
      ANI     X125  ; ËÍÁÏ¼ÐÊÖÏÂµ½Î»
      MOVP    K6 D2136
      MPS
      ANI     M90  ; 3#ÖáÆô¶¯
      SET     M90  ; 3#ÖáÆô¶¯
      MPP
      RST     B188  ; ÏòÇ°ËÍÁÏ
      MPP
      AND     B189  ; ÏòºóËÍÁÏ
      SET     Y1187  ; ÊÖ¶¯¼ÐÊÖÉý½µ·§
      SET     Y1184  ; ÊÖ¶¯¼Ð³Öµç´Å·§ONËÉ¿ªOFF¼Ð½ô
      AND     Y187  ; ËÍÁÏ¼ÐÊÖoffÉýon½µ
      ANI     X124  ; ËÍÁÏËÅ·þ¼Ð½ôÑ¹Á¦¼ì²â
      AND     X125  ; ËÍÁÏ¼ÐÊÖÏÂµ½Î»
      MOVP    K7 D2136
      MPS
      ANI     M90  ; 3#ÖáÆô¶¯
      SET     M90  ; 3#ÖáÆô¶¯
      MPP
      RST     B189  ; ÏòºóËÍÁÏ
2060  LDD=    D18 D2422  ; Öá3µ±Ç°½ø¸øÖµ / ËÍÁÏÖáÊ×³åÇ°Î»ÖÃ
      OUT     M240  ; ËÍÁÏÖáÊ×³åÇ°Î»ÖÃ±êÖ¾
2064  LDD=    D18 D2420  ; Öá3µ±Ç°½ø¸øÖµ / ËÍÁÏÖáËÅ·þ·µ»ØÎ»ÖÃ
      OUT     M241  ; ËÍÁÏÖá·µ»ØÎ»ÖÃ±êÖ¾
2068  LDP     M241  ; ËÍÁÏÖá·µ»ØÎ»ÖÃ±êÖ¾
      RST     Y1187  ; ÊÖ¶¯¼ÐÊÖÉý½µ·§
      SET     Y1184  ; ÊÖ¶¯¼Ð³Öµç´Å·§ONËÉ¿ªOFF¼Ð½ô
2071  MCR     N0
; 启动X轴
2078  LD      M50  ; 1#ÖáÆô¶¯
      PLS     M51  ; 1#ÖáÆô¶¯ÃüÁîÂö³å
2081  LD      M51  ; 1#ÖáÆô¶¯ÃüÁîÂö³å
      ANI     Y10  ; 1#Öá¶¨Î»Æô¶¯ÐÅºÅ
      ANI     X10  ; 1#ÖáÆô¶¯Íê³ÉÐÅºÅ
      ANI     X4  ; 1#ÖáM´úÂëONÐÅºÅ
      ANI     M44  ; µã¶¯
      SET     M52  ; 1#ÖáÆô¶¯ÃüÁî±£³Ö
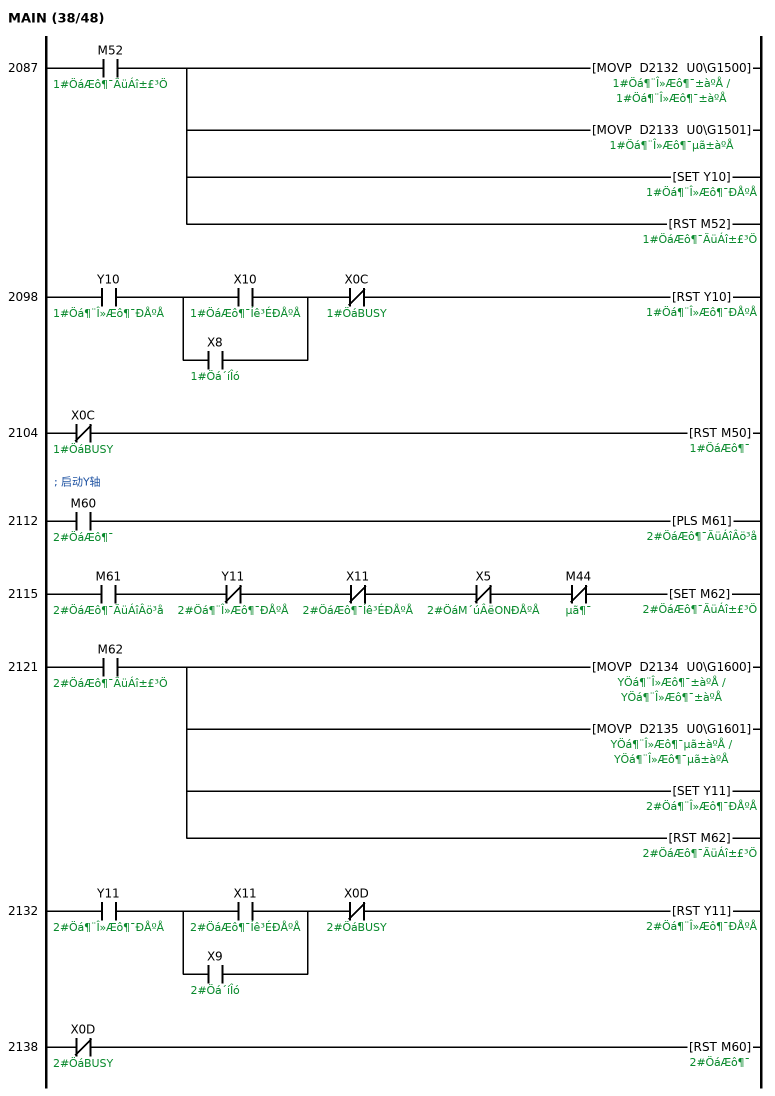
2087  LD      M52  ; 1#ÖáÆô¶¯ÃüÁî±£³Ö
      MOVP    D2132 U0\G1500  ; 1#Öá¶¨Î»Æô¶¯±àºÅ
      MOVP    D2133 U0\G1501  ; 1#Öá¶¨Î»Æô¶¯µã±àºÅ
      SET     Y10  ; 1#Öá¶¨Î»Æô¶¯ÐÅºÅ
      RST     M52  ; 1#ÖáÆô¶¯ÃüÁî±£³Ö
2098  LD      Y10  ; 1#Öá¶¨Î»Æô¶¯ÐÅºÅ
      LD      X10  ; 1#ÖáÆô¶¯Íê³ÉÐÅºÅ
      OR      X8  ; 1#Öá´íÎó
      ANB
      ANI     X0C  ; 1#ÖáBUSY
      RST     Y10  ; 1#Öá¶¨Î»Æô¶¯ÐÅºÅ
2104  LDI     X0C  ; 1#ÖáBUSY
      RST     M50  ; 1#ÖáÆô¶¯
; 启动Y轴
2112  LD      M60  ; 2#ÖáÆô¶¯
      PLS     M61  ; 2#ÖáÆô¶¯ÃüÁîÂö³å
2115  LD      M61  ; 2#ÖáÆô¶¯ÃüÁîÂö³å
      ANI     Y11  ; 2#Öá¶¨Î»Æô¶¯ÐÅºÅ
      ANI     X11  ; 2#ÖáÆô¶¯Íê³ÉÐÅºÅ
      ANI     X5  ; 2#ÖáM´úÂëONÐÅºÅ
      ANI     M44  ; µã¶¯
      SET     M62  ; 2#ÖáÆô¶¯ÃüÁî±£³Ö
2121  LD      M62  ; 2#ÖáÆô¶¯ÃüÁî±£³Ö
      MOVP    D2134 U0\G1600  ; YÖá¶¨Î»Æô¶¯±àºÅ
      MOVP    D2135 U0\G1601  ; YÖá¶¨Î»Æô¶¯µã±àºÅ / YÖá¶¨Î»Æô¶¯µã±àºÅ
      SET     Y11  ; 2#Öá¶¨Î»Æô¶¯ÐÅºÅ
      RST     M62  ; 2#ÖáÆô¶¯ÃüÁî±£³Ö
2132  LD      Y11  ; 2#Öá¶¨Î»Æô¶¯ÐÅºÅ
      LD      X11  ; 2#ÖáÆô¶¯Íê³ÉÐÅºÅ
      OR      X9  ; 2#Öá´íÎó
      ANB
      ANI     X0D  ; 2#ÖáBUSY
      RST     Y11  ; 2#Öá¶¨Î»Æô¶¯ÐÅºÅ
2138  LDI     X0D  ; 2#ÖáBUSY
      RST     M60  ; 2#ÖáÆô¶¯
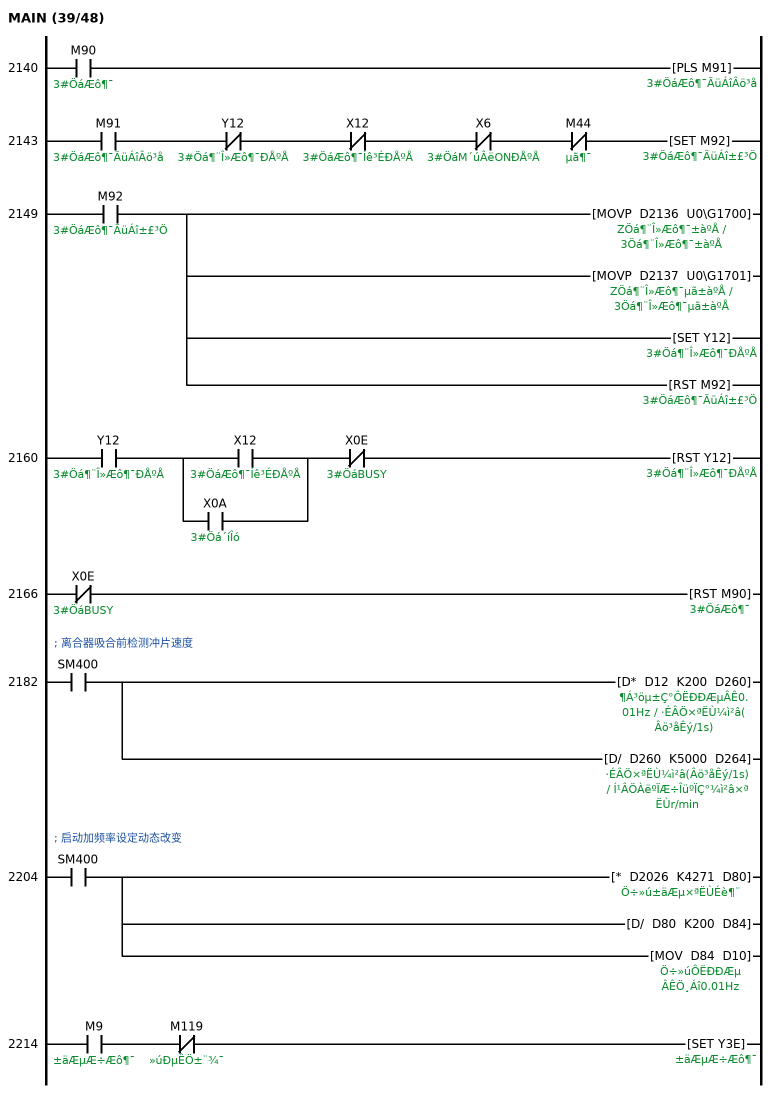
2140  LD      M90  ; 3#ÖáÆô¶¯
      PLS     M91  ; 3#ÖáÆô¶¯ÃüÁîÂö³å
2143  LD      M91  ; 3#ÖáÆô¶¯ÃüÁîÂö³å
      ANI     Y12  ; 3#Öá¶¨Î»Æô¶¯ÐÅºÅ
      ANI     X12  ; 3#ÖáÆô¶¯Íê³ÉÐÅºÅ
      ANI     X6  ; 3#ÖáM´úÂëONÐÅºÅ
      ANI     M44  ; µã¶¯
      SET     M92  ; 3#ÖáÆô¶¯ÃüÁî±£³Ö
2149  LD      M92  ; 3#ÖáÆô¶¯ÃüÁî±£³Ö
      MOVP    D2136 U0\G1700  ; 3Öá¶¨Î»Æô¶¯±àºÅ
      MOVP    D2137 U0\G1701  ; ZÖá¶¨Î»Æô¶¯µã±àºÅ / 3Öá¶¨Î»Æô¶¯µã±àºÅ
      SET     Y12  ; 3#Öá¶¨Î»Æô¶¯ÐÅºÅ
      RST     M92  ; 3#ÖáÆô¶¯ÃüÁî±£³Ö
2160  LD      Y12  ; 3#Öá¶¨Î»Æô¶¯ÐÅºÅ
      LD      X12  ; 3#ÖáÆô¶¯Íê³ÉÐÅºÅ
      OR      X0A  ; 3#Öá´íÎó
      ANB
      ANI     X0E  ; 3#ÖáBUSY
      RST     Y12  ; 3#Öá¶¨Î»Æô¶¯ÐÅºÅ
2166  LDI     X0E  ; 3#ÖáBUSY
      RST     M90  ; 3#ÖáÆô¶¯
; 离合器吸合前检测冲片速度
2182  LD      SM400
      D*      D12 K200 D260  ; ¶Á³öµ±Ç°ÔËÐÐÆµÂÊ0.01Hz / ·ÉÂÖ×ªËÙ¼ì²â(Âö³åÊý/1s)
      D/      D260 K5000 D264
; 启动加频率设定动态改变
2204  LD      SM400
      *       D2026 K4271 D80  ; Ö÷»ú±äÆµ×ªËÙÉè¶¨
      D/      D80 K200 D84
      MOV     D84 D10  ; Ö÷»úÔËÐÐÆµÂÊÖ¸Áî0.01Hz
2214  LD      M9  ; ±äÆµÆ÷Æô¶¯
      ANI     M119  ; »úÐµÊÖ±¨¾¯
      SET     Y3E  ; ±äÆµÆ÷Æô¶¯
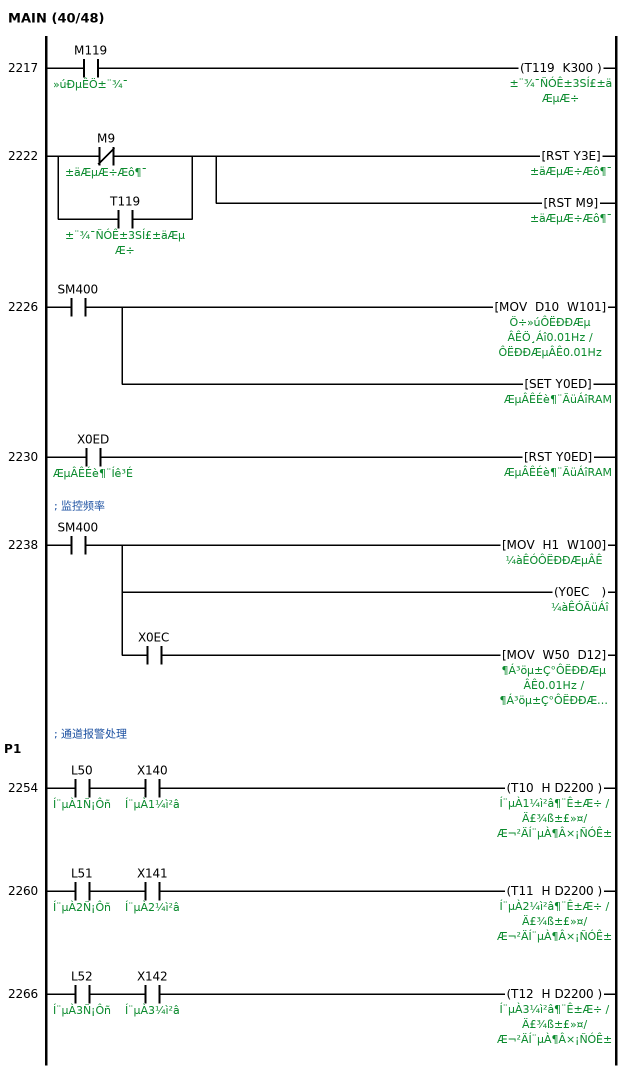
2217  LD      M119  ; »úÐµÊÖ±¨¾¯
      OUT     T119 K300  ; ±¨¾¯ÑÓÊ±3SÍ£±äÆµÆ÷
2222  LDI     M9  ; ±äÆµÆ÷Æô¶¯
      OR      T119  ; ±¨¾¯ÑÓÊ±3SÍ£±äÆµÆ÷
      RST     Y3E  ; ±äÆµÆ÷Æô¶¯
      RST     M9  ; ±äÆµÆ÷Æô¶¯
2226  LD      SM400
      MOV     D10 W101  ; ÔËÐÐÆµÂÊ0.01Hz
      SET     Y0ED  ; ÆµÂÊÉè¶¨ÃüÁîRAM
2230  LD      X0ED  ; ÆµÂÊÉè¶¨Íê³É
      RST     Y0ED  ; ÆµÂÊÉè¶¨ÃüÁîRAM
; 监控频率
2238  LD      SM400
      MOV     H1 W100  ; ¼àÊÓÔËÐÐÆµÂÊ
      OUT     Y0EC  ; ¼àÊÓÃüÁî
      AND     X0EC
      MOV     W50 D12  ; ¶Á³öµ±Ç°ÔËÐÐÆµÂÊ0.01Hz
; 通道报警处理
      P1
2254  LD      L50  ; Í¨µÀ1Ñ¡Ôñ
      AND     X140  ; Í¨µÀ1¼ì²â
      OUTH    T10 D2200  ; Í¨µÀ1¼ì²â¶¨Ê±Æ÷ / Ä£¾ß±£»¤/Æ¬²ÄÍ¨µÀ¶Â×¡ÑÓÊ±
2260  LD      L51  ; Í¨µÀ2Ñ¡Ôñ
      AND     X141  ; Í¨µÀ2¼ì²â
      OUTH    T11 D2200  ; Í¨µÀ2¼ì²â¶¨Ê±Æ÷ / Ä£¾ß±£»¤/Æ¬²ÄÍ¨µÀ¶Â×¡ÑÓÊ±
2266  LD      L52  ; Í¨µÀ3Ñ¡Ôñ
      AND     X142  ; Í¨µÀ3¼ì²â
      OUTH    T12 D2200  ; Í¨µÀ3¼ì²â¶¨Ê±Æ÷ / Ä£¾ß±£»¤/Æ¬²ÄÍ¨µÀ¶Â×¡ÑÓÊ±
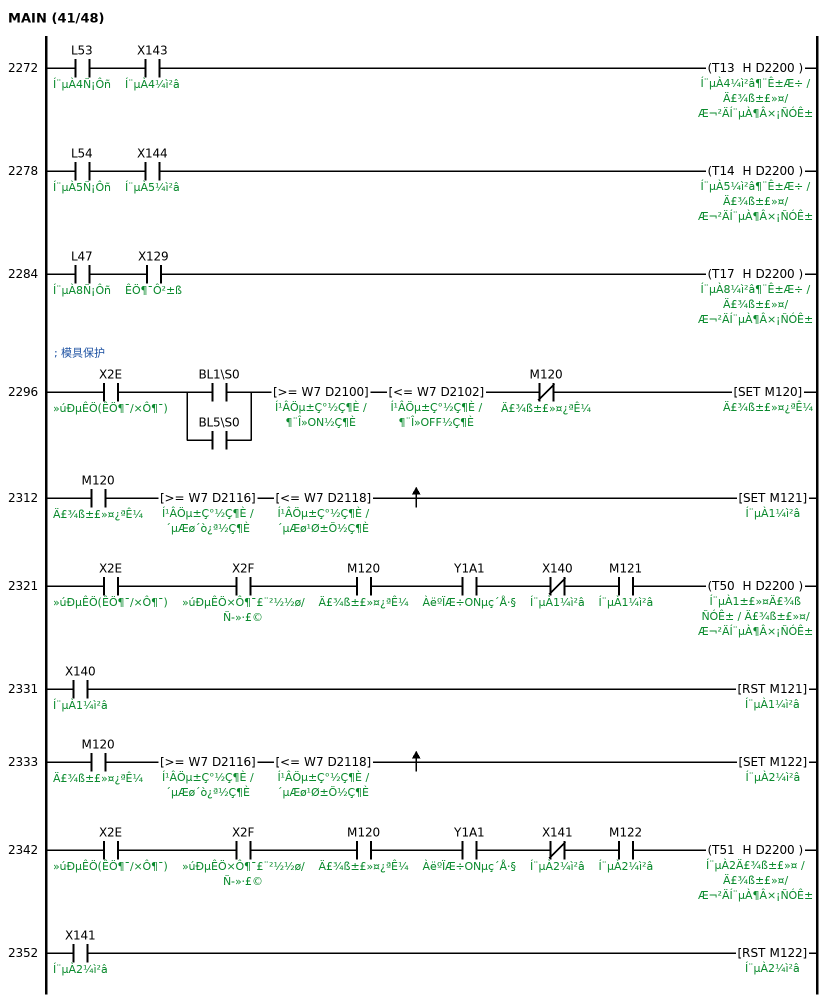
2272  LD      L53  ; Í¨µÀ4Ñ¡Ôñ
      AND     X143  ; Í¨µÀ4¼ì²â
      OUTH    T13 D2200  ; Í¨µÀ4¼ì²â¶¨Ê±Æ÷ / Ä£¾ß±£»¤/Æ¬²ÄÍ¨µÀ¶Â×¡ÑÓÊ±
2278  LD      L54  ; Í¨µÀ5Ñ¡Ôñ
      AND     X144  ; Í¨µÀ5¼ì²â
      OUTH    T14 D2200  ; Í¨µÀ5¼ì²â¶¨Ê±Æ÷ / Ä£¾ß±£»¤/Æ¬²ÄÍ¨µÀ¶Â×¡ÑÓÊ±
2284  LD      L47  ; Í¨µÀ8Ñ¡Ôñ
      AND     X129  ; ÊÖ¶¯Ô²±ß
      OUTH    T17 D2200  ; Í¨µÀ8¼ì²â¶¨Ê±Æ÷ / Ä£¾ß±£»¤/Æ¬²ÄÍ¨µÀ¶Â×¡ÑÓÊ±
; 模具保护
2296  LD      X2E  ; »úÐµÊÖ(ÊÖ¶¯/×Ô¶¯)
      LD      BL1\S0
      OR      BL5\S0
      ANB
      AND>=   W7 D2100  ; Í¹ÂÖµ±Ç°½Ç¶È / ¶¨Î»ON½Ç¶È
      AND<=   W7 D2102  ; Í¹ÂÖµ±Ç°½Ç¶È / ¶¨Î»OFF½Ç¶È
      ANI     M120  ; Ä£¾ß±£»¤¿ªÊ¼
      SET     M120  ; Ä£¾ß±£»¤¿ªÊ¼
2312  LD      M120  ; Ä£¾ß±£»¤¿ªÊ¼
      AND>=   W7 D2116  ; Í¹ÂÖµ±Ç°½Ç¶È / ´µÆø´ò¿ª½Ç¶È
      AND<=   W7 D2118  ; Í¹ÂÖµ±Ç°½Ç¶È / ´µÆø¹Ø±Õ½Ç¶È
      MEP
      SET     M121  ; Í¨µÀ1¼ì²â
2321  LD      X2E  ; »úÐµÊÖ(ÊÖ¶¯/×Ô¶¯)
      AND     X2F  ; »úÐµÊÖ×Ô¶¯£¨²½½ø/Ñ­»·£©
      AND     M120  ; Ä£¾ß±£»¤¿ªÊ¼
      AND     Y1A1  ; ÀëºÏÆ÷ONµç´Å·§
      ANI     X140  ; Í¨µÀ1¼ì²â
      AND     M121  ; Í¨µÀ1¼ì²â
      OUTH    T50 D2200  ; Í¨µÀ1±£»¤Ä£¾ßÑÓÊ± / Ä£¾ß±£»¤/Æ¬²ÄÍ¨µÀ¶Â×¡ÑÓÊ±
2331  LD      X140  ; Í¨µÀ1¼ì²â
      RST     M121  ; Í¨µÀ1¼ì²â
2333  LD      M120  ; Ä£¾ß±£»¤¿ªÊ¼
      AND>=   W7 D2116  ; Í¹ÂÖµ±Ç°½Ç¶È / ´µÆø´ò¿ª½Ç¶È
      AND<=   W7 D2118  ; Í¹ÂÖµ±Ç°½Ç¶È / ´µÆø¹Ø±Õ½Ç¶È
      MEP
      SET     M122  ; Í¨µÀ2¼ì²â
2342  LD      X2E  ; »úÐµÊÖ(ÊÖ¶¯/×Ô¶¯)
      AND     X2F  ; »úÐµÊÖ×Ô¶¯£¨²½½ø/Ñ­»·£©
      AND     M120  ; Ä£¾ß±£»¤¿ªÊ¼
      AND     Y1A1  ; ÀëºÏÆ÷ONµç´Å·§
      ANI     X141  ; Í¨µÀ2¼ì²â
      AND     M122  ; Í¨µÀ2¼ì²â
      OUTH    T51 D2200  ; Í¨µÀ2Ä£¾ß±£»¤ / Ä£¾ß±£»¤/Æ¬²ÄÍ¨µÀ¶Â×¡ÑÓÊ±
2352  LD      X141  ; Í¨µÀ2¼ì²â
      RST     M122  ; Í¨µÀ2¼ì²â
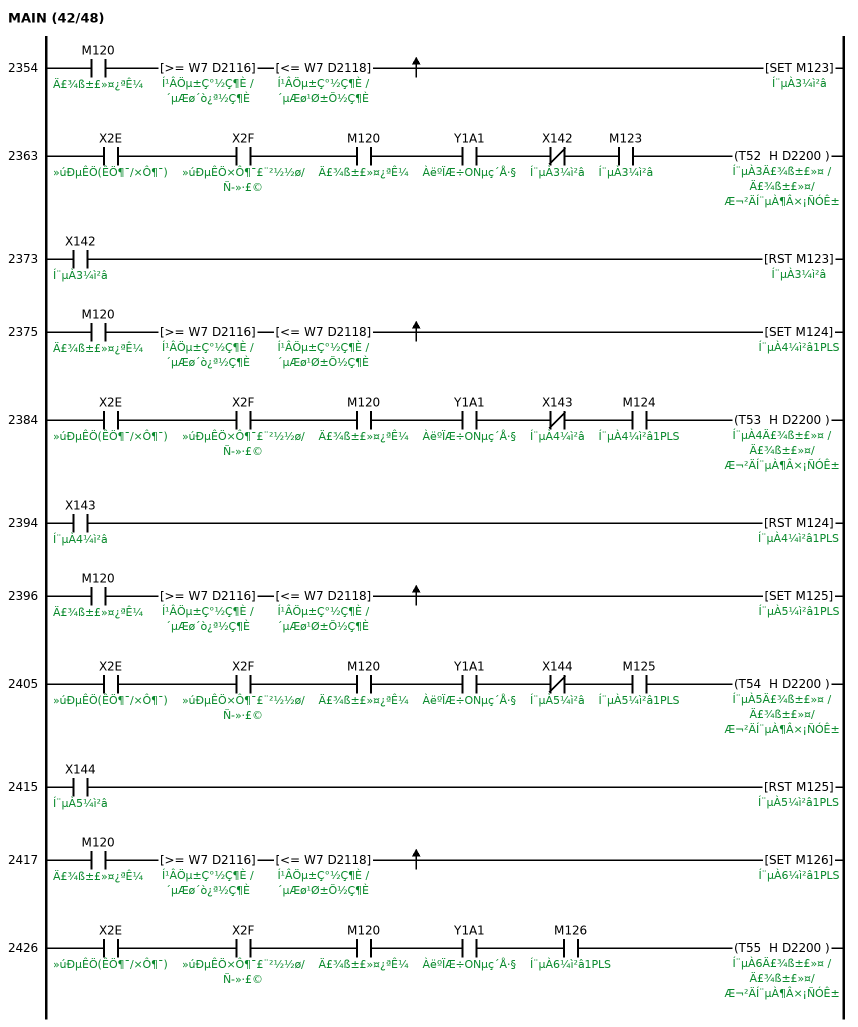
2354  LD      M120  ; Ä£¾ß±£»¤¿ªÊ¼
      AND>=   W7 D2116  ; Í¹ÂÖµ±Ç°½Ç¶È / ´µÆø´ò¿ª½Ç¶È
      AND<=   W7 D2118  ; Í¹ÂÖµ±Ç°½Ç¶È / ´µÆø¹Ø±Õ½Ç¶È
      MEP
      SET     M123  ; Í¨µÀ3¼ì²â
2363  LD      X2E  ; »úÐµÊÖ(ÊÖ¶¯/×Ô¶¯)
      AND     X2F  ; »úÐµÊÖ×Ô¶¯£¨²½½ø/Ñ­»·£©
      AND     M120  ; Ä£¾ß±£»¤¿ªÊ¼
      AND     Y1A1  ; ÀëºÏÆ÷ONµç´Å·§
      ANI     X142  ; Í¨µÀ3¼ì²â
      AND     M123  ; Í¨µÀ3¼ì²â
      OUTH    T52 D2200  ; Í¨µÀ3Ä£¾ß±£»¤ / Ä£¾ß±£»¤/Æ¬²ÄÍ¨µÀ¶Â×¡ÑÓÊ±
2373  LD      X142  ; Í¨µÀ3¼ì²â
      RST     M123  ; Í¨µÀ3¼ì²â
2375  LD      M120  ; Ä£¾ß±£»¤¿ªÊ¼
      AND>=   W7 D2116  ; Í¹ÂÖµ±Ç°½Ç¶È / ´µÆø´ò¿ª½Ç¶È
      AND<=   W7 D2118  ; Í¹ÂÖµ±Ç°½Ç¶È / ´µÆø¹Ø±Õ½Ç¶È
      MEP
      SET     M124  ; Í¨µÀ4¼ì²â1PLS
2384  LD      X2E  ; »úÐµÊÖ(ÊÖ¶¯/×Ô¶¯)
      AND     X2F  ; »úÐµÊÖ×Ô¶¯£¨²½½ø/Ñ­»·£©
      AND     M120  ; Ä£¾ß±£»¤¿ªÊ¼
      AND     Y1A1  ; ÀëºÏÆ÷ONµç´Å·§
      ANI     X143  ; Í¨µÀ4¼ì²â
      AND     M124  ; Í¨µÀ4¼ì²â1PLS
      OUTH    T53 D2200  ; Í¨µÀ4Ä£¾ß±£»¤ / Ä£¾ß±£»¤/Æ¬²ÄÍ¨µÀ¶Â×¡ÑÓÊ±
2394  LD      X143  ; Í¨µÀ4¼ì²â
      RST     M124  ; Í¨µÀ4¼ì²â1PLS
2396  LD      M120  ; Ä£¾ß±£»¤¿ªÊ¼
      AND>=   W7 D2116  ; Í¹ÂÖµ±Ç°½Ç¶È / ´µÆø´ò¿ª½Ç¶È
      AND<=   W7 D2118  ; Í¹ÂÖµ±Ç°½Ç¶È / ´µÆø¹Ø±Õ½Ç¶È
      MEP
      SET     M125  ; Í¨µÀ5¼ì²â1PLS
2405  LD      X2E  ; »úÐµÊÖ(ÊÖ¶¯/×Ô¶¯)
      AND     X2F  ; »úÐµÊÖ×Ô¶¯£¨²½½ø/Ñ­»·£©
      AND     M120  ; Ä£¾ß±£»¤¿ªÊ¼
      AND     Y1A1  ; ÀëºÏÆ÷ONµç´Å·§
      ANI     X144  ; Í¨µÀ5¼ì²â
      AND     M125  ; Í¨µÀ5¼ì²â1PLS
      OUTH    T54 D2200  ; Í¨µÀ5Ä£¾ß±£»¤ / Ä£¾ß±£»¤/Æ¬²ÄÍ¨µÀ¶Â×¡ÑÓÊ±
2415  LD      X144  ; Í¨µÀ5¼ì²â
      RST     M125  ; Í¨µÀ5¼ì²â1PLS
2417  LD      M120  ; Ä£¾ß±£»¤¿ªÊ¼
      AND>=   W7 D2116  ; Í¹ÂÖµ±Ç°½Ç¶È / ´µÆø´ò¿ª½Ç¶È
      AND<=   W7 D2118  ; Í¹ÂÖµ±Ç°½Ç¶È / ´µÆø¹Ø±Õ½Ç¶È
      MEP
      SET     M126  ; Í¨µÀ6¼ì²â1PLS
2426  LD      X2E  ; »úÐµÊÖ(ÊÖ¶¯/×Ô¶¯)
      AND     X2F  ; »úÐµÊÖ×Ô¶¯£¨²½½ø/Ñ­»·£©
      AND     M120  ; Ä£¾ß±£»¤¿ªÊ¼
      AND     Y1A1  ; ÀëºÏÆ÷ONµç´Å·§
      AND     M126  ; Í¨µÀ6¼ì²â1PLS
      OUTH    T55 D2200  ; Í¨µÀ6Ä£¾ß±£»¤ / Ä£¾ß±£»¤/Æ¬²ÄÍ¨µÀ¶Â×¡ÑÓÊ±
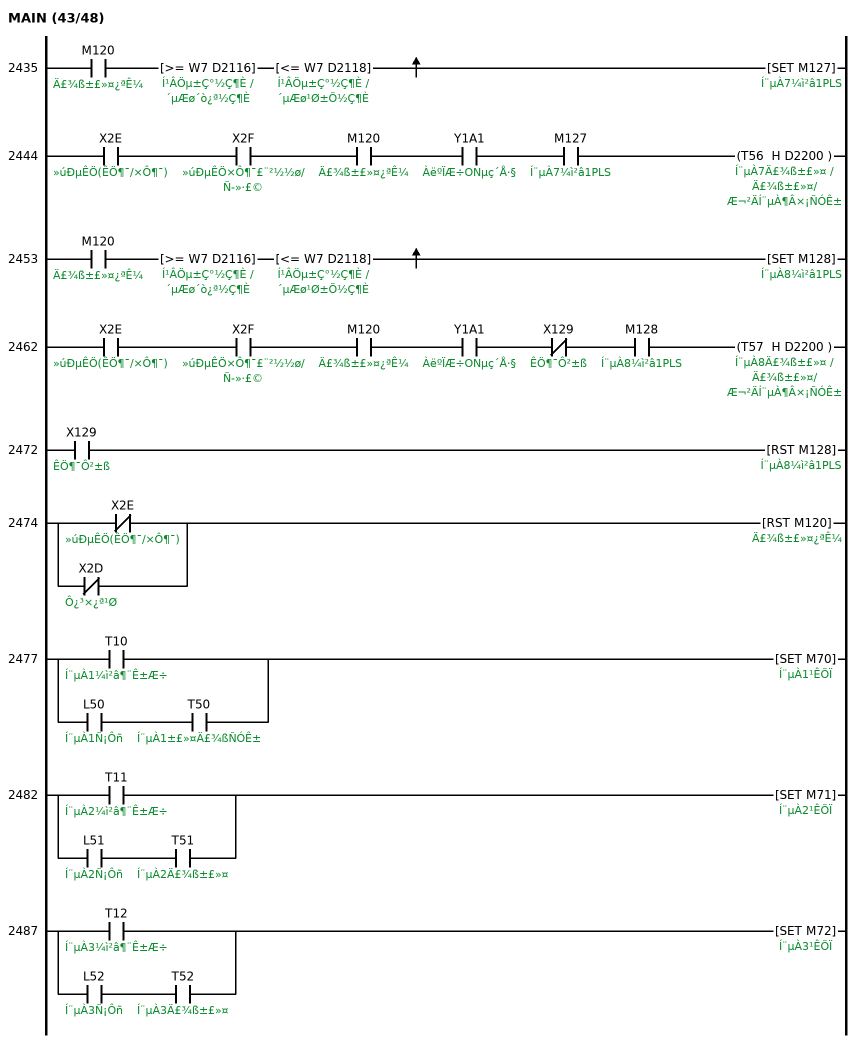
2435  LD      M120  ; Ä£¾ß±£»¤¿ªÊ¼
      AND>=   W7 D2116  ; Í¹ÂÖµ±Ç°½Ç¶È / ´µÆø´ò¿ª½Ç¶È
      AND<=   W7 D2118  ; Í¹ÂÖµ±Ç°½Ç¶È / ´µÆø¹Ø±Õ½Ç¶È
      MEP
      SET     M127  ; Í¨µÀ7¼ì²â1PLS
2444  LD      X2E  ; »úÐµÊÖ(ÊÖ¶¯/×Ô¶¯)
      AND     X2F  ; »úÐµÊÖ×Ô¶¯£¨²½½ø/Ñ­»·£©
      AND     M120  ; Ä£¾ß±£»¤¿ªÊ¼
      AND     Y1A1  ; ÀëºÏÆ÷ONµç´Å·§
      AND     M127  ; Í¨µÀ7¼ì²â1PLS
      OUTH    T56 D2200  ; Í¨µÀ7Ä£¾ß±£»¤ / Ä£¾ß±£»¤/Æ¬²ÄÍ¨µÀ¶Â×¡ÑÓÊ±
2453  LD      M120  ; Ä£¾ß±£»¤¿ªÊ¼
      AND>=   W7 D2116  ; Í¹ÂÖµ±Ç°½Ç¶È / ´µÆø´ò¿ª½Ç¶È
      AND<=   W7 D2118  ; Í¹ÂÖµ±Ç°½Ç¶È / ´µÆø¹Ø±Õ½Ç¶È
      MEP
      SET     M128  ; Í¨µÀ8¼ì²â1PLS
2462  LD      X2E  ; »úÐµÊÖ(ÊÖ¶¯/×Ô¶¯)
      AND     X2F  ; »úÐµÊÖ×Ô¶¯£¨²½½ø/Ñ­»·£©
      AND     M120  ; Ä£¾ß±£»¤¿ªÊ¼
      AND     Y1A1  ; ÀëºÏÆ÷ONµç´Å·§
      ANI     X129  ; ÊÖ¶¯Ô²±ß
      AND     M128  ; Í¨µÀ8¼ì²â1PLS
      OUTH    T57 D2200  ; Í¨µÀ8Ä£¾ß±£»¤ / Ä£¾ß±£»¤/Æ¬²ÄÍ¨µÀ¶Â×¡ÑÓÊ±
2472  LD      X129  ; ÊÖ¶¯Ô²±ß
      RST     M128  ; Í¨µÀ8¼ì²â1PLS
2474  LDI     X2E  ; »úÐµÊÖ(ÊÖ¶¯/×Ô¶¯)
      ORI     X2D  ; Ô¿³×¿ª¹Ø
      RST     M120  ; Ä£¾ß±£»¤¿ªÊ¼
2477  LD      T10  ; Í¨µÀ1¼ì²â¶¨Ê±Æ÷
      LD      L50  ; Í¨µÀ1Ñ¡Ôñ
      AND     T50  ; Í¨µÀ1±£»¤Ä£¾ßÑÓÊ±
      ORB
      SET     M70  ; Í¨µÀ1¹ÊÕÏ
2482  LD      T11  ; Í¨µÀ2¼ì²â¶¨Ê±Æ÷
      LD      L51  ; Í¨µÀ2Ñ¡Ôñ
      AND     T51  ; Í¨µÀ2Ä£¾ß±£»¤
      ORB
      SET     M71  ; Í¨µÀ2¹ÊÕÏ
2487  LD      T12  ; Í¨µÀ3¼ì²â¶¨Ê±Æ÷
      LD      L52  ; Í¨µÀ3Ñ¡Ôñ
      AND     T52  ; Í¨µÀ3Ä£¾ß±£»¤
      ORB
      SET     M72  ; Í¨µÀ3¹ÊÕÏ
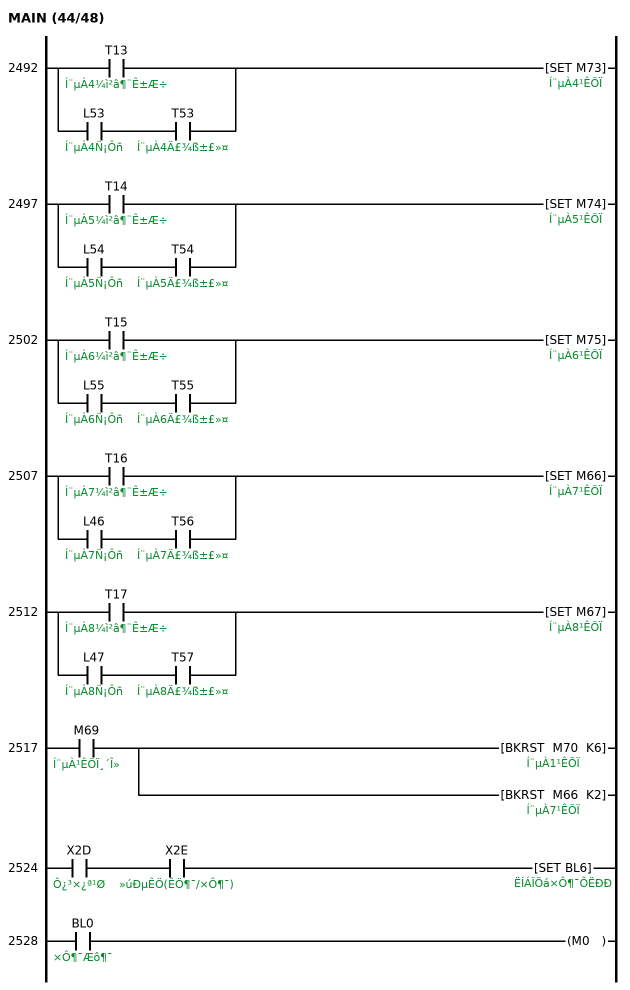
2492  LD      T13  ; Í¨µÀ4¼ì²â¶¨Ê±Æ÷
      LD      L53  ; Í¨µÀ4Ñ¡Ôñ
      AND     T53  ; Í¨µÀ4Ä£¾ß±£»¤
      ORB
      SET     M73  ; Í¨µÀ4¹ÊÕÏ
2497  LD      T14  ; Í¨µÀ5¼ì²â¶¨Ê±Æ÷
      LD      L54  ; Í¨µÀ5Ñ¡Ôñ
      AND     T54  ; Í¨µÀ5Ä£¾ß±£»¤
      ORB
      SET     M74  ; Í¨µÀ5¹ÊÕÏ
2502  LD      T15  ; Í¨µÀ6¼ì²â¶¨Ê±Æ÷
      LD      L55  ; Í¨µÀ6Ñ¡Ôñ
      AND     T55  ; Í¨µÀ6Ä£¾ß±£»¤
      ORB
      SET     M75  ; Í¨µÀ6¹ÊÕÏ
2507  LD      T16  ; Í¨µÀ7¼ì²â¶¨Ê±Æ÷
      LD      L46  ; Í¨µÀ7Ñ¡Ôñ
      AND     T56  ; Í¨µÀ7Ä£¾ß±£»¤
      ORB
      SET     M66  ; Í¨µÀ7¹ÊÕÏ
2512  LD      T17  ; Í¨µÀ8¼ì²â¶¨Ê±Æ÷
      LD      L47  ; Í¨µÀ8Ñ¡Ôñ
      AND     T57  ; Í¨µÀ8Ä£¾ß±£»¤
      ORB
      SET     M67  ; Í¨µÀ8¹ÊÕÏ
2517  LD      M69  ; Í¨µÀ¹ÊÕÏ¸´Î»
      BKRST   M70 K6
      BKRST   M66 K2
2524  LD      X2D  ; Ô¿³×¿ª¹Ø
      AND     X2E  ; »úÐµÊÖ(ÊÖ¶¯/×Ô¶¯)
      SET     BL6  ; ËÍÁÏÖá×Ô¶¯ÔËÐÐ
2528  LD      BL0  ; ×Ô¶¯Æô¶¯
      OUT     M0
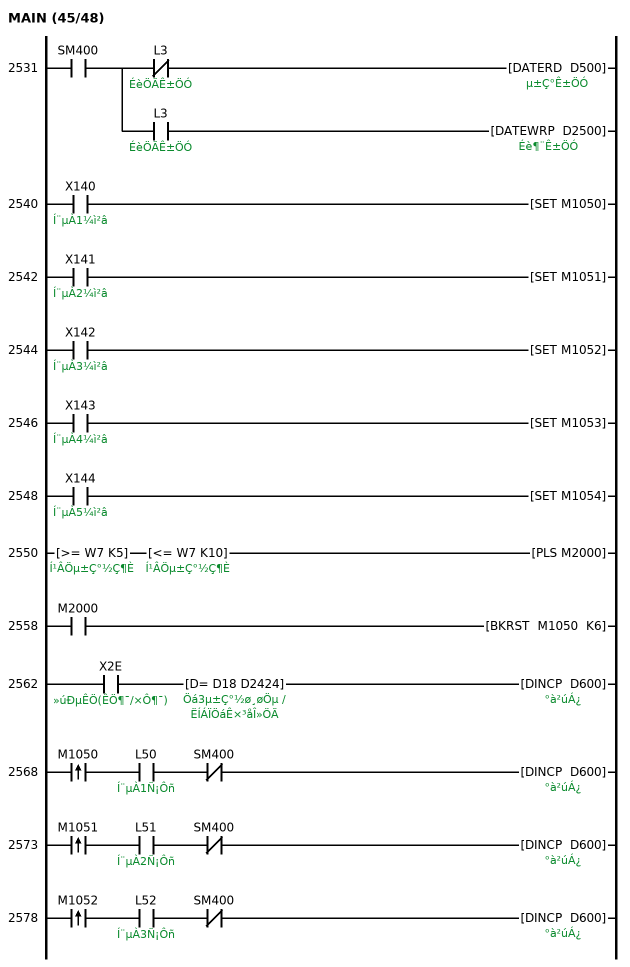
2531  LD      SM400
      MPS
      ANI     L3  ; ÉèÖÃÊ±ÖÓ
      DATERD  D500  ; µ±Ç°Ê±ÖÓ
      MPP
      AND     L3  ; ÉèÖÃÊ±ÖÓ
      DATEWRP D2500  ; Éè¶¨Ê±ÖÓ
2540  LD      X140  ; Í¨µÀ1¼ì²â
      SET     M1050
2542  LD      X141  ; Í¨µÀ2¼ì²â
      SET     M1051
2544  LD      X142  ; Í¨µÀ3¼ì²â
      SET     M1052
2546  LD      X143  ; Í¨µÀ4¼ì²â
      SET     M1053
2548  LD      X144  ; Í¨µÀ5¼ì²â
      SET     M1054
2550  LD>=    W7 K5  ; Í¹ÂÖµ±Ç°½Ç¶È
      AND<=   W7 K10  ; Í¹ÂÖµ±Ç°½Ç¶È
      PLS     M2000
2558  LD      M2000
      BKRST   M1050 K6
2562  LD      X2E  ; »úÐµÊÖ(ÊÖ¶¯/×Ô¶¯)
      ANDD=   D18 D2424  ; Öá3µ±Ç°½ø¸øÖµ / ËÍÁÏÖáÊ×³åÎ»ÖÃ
      DINCP   D600  ; °à²úÁ¿
2568  LDP     M1050
      AND     L50  ; Í¨µÀ1Ñ¡Ôñ
      ANI     SM400
      DINCP   D600
2573  LDP     M1051
      AND     L51  ; Í¨µÀ2Ñ¡Ôñ
      ANI     SM400
      DINCP   D600
2578  LDP     M1052
      AND     L52  ; Í¨µÀ3Ñ¡Ôñ
      ANI     SM400
      DINCP   D600
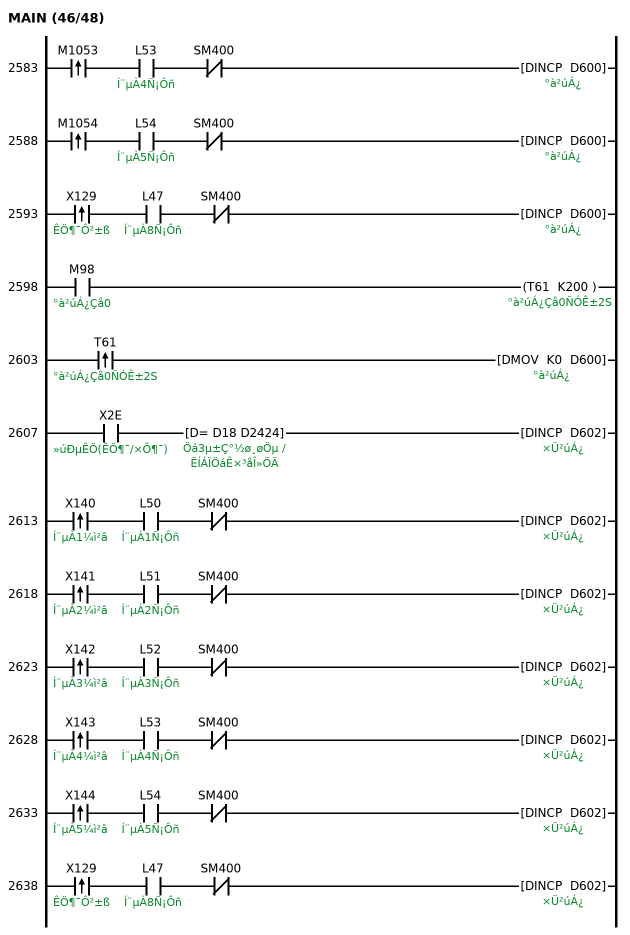
2583  LDP     M1053
      AND     L53  ; Í¨µÀ4Ñ¡Ôñ
      ANI     SM400
      DINCP   D600
2588  LDP     M1054
      AND     L54  ; Í¨µÀ5Ñ¡Ôñ
      ANI     SM400
      DINCP   D600
2593  LDP     X129  ; ÊÖ¶¯Ô²±ß
      AND     L47  ; Í¨µÀ8Ñ¡Ôñ
      ANI     SM400
      DINCP   D600
2598  LD      M98  ; °à²úÁ¿Çå0
      OUT     T61 K200  ; °à²úÁ¿Çå0ÑÓÊ±2S
2603  LDP     T61  ; °à²úÁ¿Çå0ÑÓÊ±2S
      DMOV    K0 D600
2607  LD      X2E  ; »úÐµÊÖ(ÊÖ¶¯/×Ô¶¯)
      ANDD=   D18 D2424  ; Öá3µ±Ç°½ø¸øÖµ / ËÍÁÏÖáÊ×³åÎ»ÖÃ
      DINCP   D602  ; ×Ü²úÁ¿
2613  LDP     X140  ; Í¨µÀ1¼ì²â
      AND     L50  ; Í¨µÀ1Ñ¡Ôñ
      ANI     SM400
      DINCP   D602
2618  LDP     X141  ; Í¨µÀ2¼ì²â
      AND     L51  ; Í¨µÀ2Ñ¡Ôñ
      ANI     SM400
      DINCP   D602
2623  LDP     X142  ; Í¨µÀ3¼ì²â
      AND     L52  ; Í¨µÀ3Ñ¡Ôñ
      ANI     SM400
      DINCP   D602
2628  LDP     X143  ; Í¨µÀ4¼ì²â
      AND     L53  ; Í¨µÀ4Ñ¡Ôñ
      ANI     SM400
      DINCP   D602
2633  LDP     X144  ; Í¨µÀ5¼ì²â
      AND     L54  ; Í¨µÀ5Ñ¡Ôñ
      ANI     SM400
      DINCP   D602
2638  LDP     X129  ; ÊÖ¶¯Ô²±ß
      AND     L47  ; Í¨µÀ8Ñ¡Ôñ
      ANI     SM400
      DINCP   D602
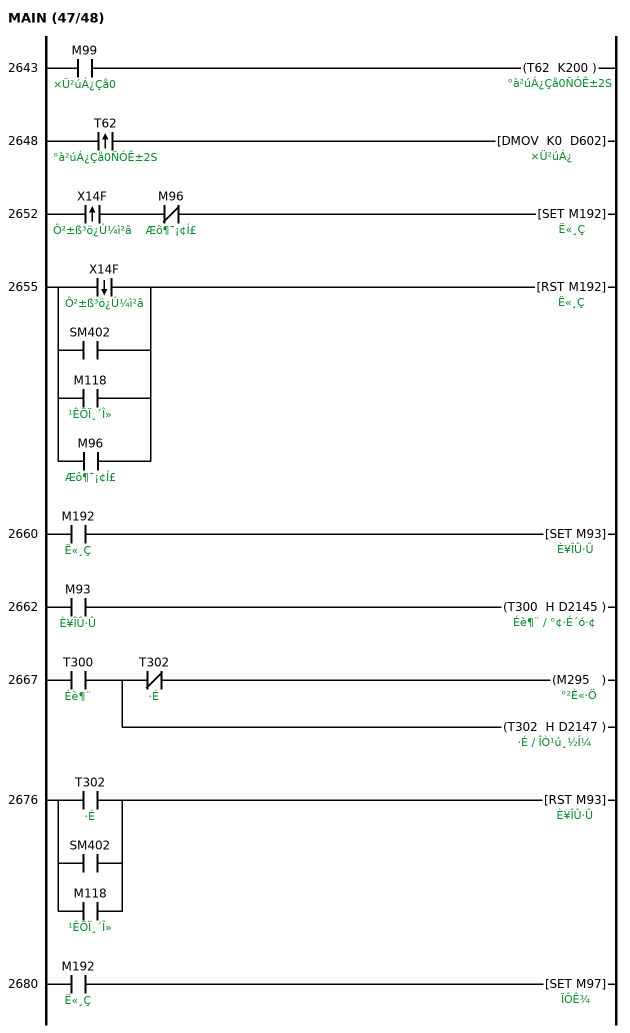
2643  LD      M99  ; ×Ü²úÁ¿Çå0
      OUT     T62 K200  ; °à²úÁ¿Çå0ÑÓÊ±2S
2648  LDP     T62  ; °à²úÁ¿Çå0ÑÓÊ±2S
      DMOV    K0 D602
2652  LDP     X14F  ; Ô²±ß³ö¿Ú¼ì²â
      ANI     M96  ; Æô¶¯¡¢Í£
      SET     M192  ; Ë«¸Ç
2655  LDF     X14F  ; Ô²±ß³ö¿Ú¼ì²â
      OR      SM402
      OR      M118  ; ¹ÊÕÏ¸´Î»
      OR      M96  ; Æô¶¯¡¢Í£
      RST     M192  ; Ë«¸Ç
2660  LD      M192  ; Ë«¸Ç
      SET     M93  ; È¥ÎÛ·Û
2662  LD      M93  ; È¥ÎÛ·Û
      OUTH    T300 D2145  ; Éè¶¨ / °¢·É´ó·¢
2667  LD      T300  ; Éè¶¨
      MPS
      ANI     T302  ; ·É
      OUT     M295  ; °²È«·Ö
      MPP
      OUTH    T302 D2147  ; ·É / ÎÒ¹ú¸½Í¼
2676  LD      T302  ; ·É
      OR      SM402
      OR      M118  ; ¹ÊÕÏ¸´Î»
      RST     M93  ; È¥ÎÛ·Û
2680  LD      M192  ; Ë«¸Ç
      SET     M97  ; ÏÔÊ¾
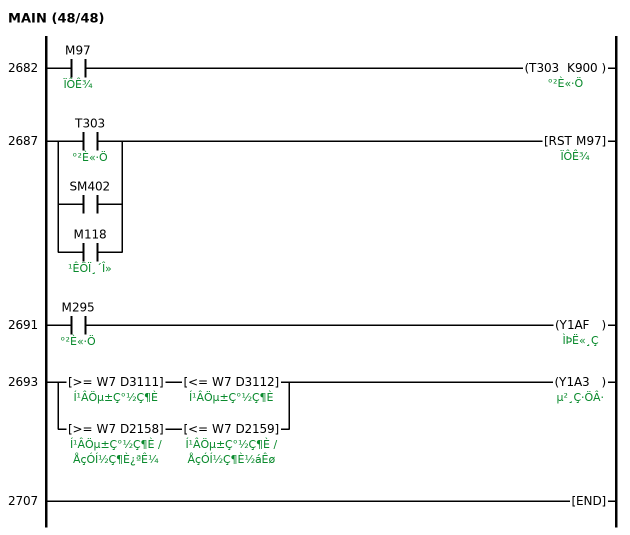
2682  LD      M97  ; ÏÔÊ¾
      OUT     T303 K900  ; °²È«·Ö
2687  LD      T303  ; °²È«·Ö
      OR      SM402
      OR      M118  ; ¹ÊÕÏ¸´Î»
      RST     M97  ; ÏÔÊ¾
2691  LD      M295  ; °²È«·Ö
      OUT     Y1AF  ; ÌÞË«¸Ç
2693  LD>=    W7 D3111  ; Í¹ÂÖµ±Ç°½Ç¶È
      AND<=   W7 D3112  ; Í¹ÂÖµ±Ç°½Ç¶È
      LD>=    W7 D2158  ; Í¹ÂÖµ±Ç°½Ç¶È / ÅçÓÍ½Ç¶È¿ªÊ¼
      AND<=   W7 D2159  ; Í¹ÂÖµ±Ç°½Ç¶È / ÅçÓÍ½Ç¶È½áÊø
      ORB
      OUT     Y1A3  ; µ²¸Ç·ÖÂ·
2707  END
END_PROGRAM

// 7 SFC block(s) not rendered

// device comments not shown above
X61  ; ¾øµØÖµ±àÂëÆ÷2
X62  ; ¾øµØÖµ±àÂëÆ÷3
X63  ; ¾øµØÖµ±àÂëÆ÷4
X64  ; ¾øµØÖµ±àÂëÆ÷5
X65  ; ¾øµØÖµ±àÂëÆ÷6
X66  ; ¾øµØÖµ±àÂëÆ÷7
X67  ; ¾øµØÖµ±àÂëÆ÷8
X68  ; ¾øµØÖµ±àÂëÆ÷9
X69  ; ¾øµØÖµ±àÂëÆ÷10
X103  ; ·ÖÕÅºóÎüÉÏ1µ½Î»
X104  ; ·ÖÕÅºóÎüÉÏ2µ½Î»
X105  ; ·ÖÕÅÇ°ÎüÉÏ1µ½Î»
X106  ; ·ÖÕÅÇ°ÎüÉÏ2µ½Î»
X107  ; ·ÖÕÅÇ°ÎüÉÏ3µ½Î»
X108  ; ·ÖÕÅËÍÁÏµ½Î»
X109  ; ·ÖÕÅËÍÁÏ¸´Î»
X10D  ; ·ÖÕÅºóÎüµç´Å·§ÏÂµ½Î»
X10F  ; ·ÖÕÅÇ°Îüµç´Å·§ÏÂµ½Î»
X120  ; ¹¤×÷Ì¨ÂäÁÏµ½Î»
X122  ; ¹¤×÷Ì¨ÓÒºó¶¨Î»
X123  ; ¹¤×÷Ì¨²â¶¨Î»
X127  ; ×¥ÊÖºÏÂ£Ñ¹Á¦¼ì²â
X128  ; ¹¤×÷Ì¨Ì§ÉýÏÂµ½Î»
X12A  ; ¹¤×÷Ì¨ËÍÁÏµ½Ç°¼ì²â
X12C  ; ¹¤×÷Ì¨×óºó¶¨Î»
X14B  ; ÅÅ·ÏÁÏÉÏÏÞÎ»
Y3F  ; ±äÆµÆ÷¸´Î»
Y0E0  ; ±äÆµÕý×ªÆô¶¯
Y1032  ; Õæ¿Õ±Ãµç»úÊÖ¶¯
Y1034  ; Ö÷Í¨·çµç»úÊÖ¶¯
Y103A  ; Ô²±ßµç»ú2ÊÖ¶¯
Y1181  ; ÊÖ¶¯ÂäÁÏÎüµç´Å·§
Y1182  ; ÊÖ¶¯Ïòºó¶¨Î»µç´Å·§
Y1183  ; ÊÖ¶¯Ïò²à¶¨Î»µç´Å·§
Y11A3  ; ÊÖ¶¯ÅçÓÍ
M3  ; ÔÊÐíÊÖ¶¯¿ªËÅ·þ
M7  ; ÀëºÏÆ÷ON/OFFÖ¸Áî£¨ÊÖ¶¯Ê±£©
M8  ; ÀëºÏÆ÷ON/OFF(×Ô¶¯Æô¶¯)
M100  ; Ç¿ÖÆÆô¶¯·ÖÕÅ»ú¹¹
M112  ; tuy
M115  ; ËÍÆ¬ÑÓÊ±
M190  ; ÌáÇ°Æô¶¯Æ¬ÁÏÌ§Éý
M250  ; ÖÐÎÄ
M251  ; Ó¢ÎÄ
M412  ; 1s
M1001  ; Í¹ÂÖµ±Ç°Öµ<=ÀëºÏÆ÷OFF½Ç¶È
M1011  ; Ê×³åÇ°Î»ÖÃ
M6008  ; Ä£ÄâÅçÓÍÐÅºÅ
L0  ; 60¶È/90¶È  OFF·½¿×
L20  ; XÖáÆæÊýÅÅÒÆ¶¯·½Ïò
L21  ; XÖáÅ¼ÊýÅÅÒÆ¶¯·½Ïò
L22  ; XÖá¼Äµ½Å¼ÒÆ¶¯·½Ïò
L23  ; XÖáÅ¼µ½¼ÄÒÆ¶¯·½Ïò
L42  ; ¶¥ÁÏÔÊÐí/½ûÖ¹
L57  ; Ö÷Í¨·çµç»úÔÊÐí/½ûÖ¹
T5  ; ÅçÓÍÊ±¼ä
T6  ; ÓÐÁÏ¼ì²âºóÑÓÊ±1S(È·±£ÁÏÎÈ¶¨)
T7  ; ËÍÆ¬ÑÓÊ±
T8  ; ºó¶¨Î»µ½ÑÓÊ±100ms
T20  ; ÎüÁÏÑÓÊ±(È·±£ÁÏÎü×¡)
T21  ; ºó¶¨Î»£¬²â¶¨Î»½áÊøÑÓÊ±100ms
T22  ; µ²ÁÏ¸×ÂäÏÂºÍ¼Ð½ôÑÓÊ±100ms
T24  ; ¶¨Î»¼ÐÊÖµ½Î»£¬¿ÉÒÔËÍÁÏÑÓÊ±100ms
T30  ; ÑÓÊ±
T33  ; ¼Ð½ôÑÓÊ±
T43  ; ·­°åONÑÓÊ±100ms
T45  ; Ê×³åÆô¶¯ÑÓ³Ù°Ú¶¯Ê±¼ä
T88  ; Ë«¸Ç
T92  ; ¹¤×÷Ì¨ÓÐÁÏÑÓÊ±
D36  ; XÖáµ±Ç°Æô¶¯±àºÅ
D37  ; YÖáµ±Ç°Æô¶¯±àºÅ
D39  ; Öá1µ±Ç°×´Ì¬
D40  ; Öá2µ±Ç°×´Ì¬
D100  ; XÖá0¶È¶¨Î»³¤¶ÈD+¼ä¸ô
D102  ; XÖá0¶È¶¨Î»³¤¶È£¨D+¼ä¸ô£©¸¡µãÊý
D104  ; ¶¨Î»½Ç¶È×ª»»¸¡µãÊý
D106  ; ¶¨Î»½Ç¶È×ª»»Îª»¡¶È
D108  ; SIN60¶È
D110  ; COS60¶È
D112  ; YÖá¶¨Î»³¤¶È¸¡µãÊý
D114  ; XÖá¶¨Î»³¤¶È£¨²î²¹£©¸¡µãÊý
D118  ; XÖá¶¨Î»³¤¶È²î²¹£¨D+¼ä¸ô£©COS60
D120  ; D/2
D124  ; Ye
D126  ; µÚÒ»³åÇ°¶¨Î»³¤¶ÈYo+Ye
D136  ; m-1ÅÅ¸¡µãÊý
D138  ; mÅÅ¸¡µãÊý
D140  ; mÅÅ
D150  ; n-1ÁÐ¸¡µãÊý
D152  ; nÁÐ¸¡µãÊý
D154  ; nÁÐ
D156  ; ³åÆ¬Ö±¾¶D¸¡µãÊý
D158  ; mÅÅ¸¡µãÊý
D160  ; nÁÐ¸¡µãÊý
D162  ; Æ¬²Ä³¤¶È¸¡µãÊý
D164  ; Æ¬²Ä¿í¶È¸¡µãÊý
D182  ; ³åÆ¬Ð§ÂÊ
D184  ; XÖá0¶È¶¨Î»³¤¶È¸ºÖµ-£¨D+¼ä¸ô£©
D188  ; XÖá¶¨Î»³¤¶È£¨²î²¹£©¸ºÖµ
D192  ; l-L
D194  ; l-L+l1
D206  ; 1Â·¾¶¶¨Î»X2
D208  ; 1Â·¾¶¶¨Î»X3
D210  ; 1Â·¾¶¶¨Î»X4
D212  ; 2Â·¾¶¶¨Î»X2
D214  ; 2Â·¾¶¶¨Î»X3
D216  ; 2Â·¾¶¶¨Î»X4
D218  ; µÚÈýÂ·¾¶µÚ2¶¨Î»
D220  ; µÚÈýÂ·¾¶µÚ3¶¨Î»
D222  ; µÚÈýÂ·¾¶µÚ4¶¨Î»
D224  ; µÚÈýÂ·¾¶µÚ5¶¨Î»
D226  ; µÚÈýÂ·¾¶µÚ6¶¨Î»
D228  ; µÚ1£¬2Â·¾¶×î´óÐÐ³Ì
D240  ; 3Â·¾¶Ê×³åÇ°¶¨Î»Î»ÖÃ
D244  ; 1Â·¾¶¶¨Î»X1
D246  ; 2Â·¾¶¶¨Î»X1
D248  ; 3Â·¾¶¶¨Î»X1
D262  ; ·ÉÂÖ×ªËÙ¼ì²â(Âö³åÊý/1mim)
D2028  ; XÖáÆæÊýÅÅÒÆ¶¯´ÎÊý
D2030  ; XÖáÅ¼ÊýÅÅÒÆ¶¯´ÎÊý
D2038  ; YoµÚÒ»³åÄ£¾ß³¤¶È²ÎÊý
D2044  ; Æ¬²Ä¿í¶È
D2046  ; Æ¬²Ä³¤¶ÈL
D2050  ; ³å¼¸ÅÅ¿ªÊ¼ÏòÇ°ËÍÁÏ
D2108  ; ÌÞ·ÏON½Ç¶È
D2110  ; ÌÞ·ÏOFF½Ç¶È
D2138  ; XÖáÆæÊýÅÅÆ½ÒÆµ±Ç°Ñ­»·´ÎÊý
D2140  ; XÖáÅ¼ÊýÅÅÆ½ÒÆµ±Ç°Ñ­»·´ÎÊý
D2142  ; Ñ­»·XÖá¶¨Î»Î»ÖÃ
D2150  ; µ±Ç°Ñ­»·´ÎÊý
D2152  ; Ñ­»·YÖá¶¨Î»Î»ÖÃ
